// TwinCAT 3 PLC project IntelligenteWZM_PLCProject
// ProgramVersion: 3.1.4022.4
// libraries:
//   Tc2_Standard, * (Beckhoff Automation GmbH)
//   Tc2_System, * (Beckhoff Automation GmbH)
//   Tc2_Utilities, * (Beckhoff Automation GmbH)
//   Tc3_CM, * (Beckhoff Automation GmbH)
//   Tc3_CM_Base, * (Beckhoff Automation GmbH)
//   Tc3_Module, * (Beckhoff Automation GmbH)
//   Tc3_MultiArray, * (Beckhoff Automation GmbH)
//   VisuDialogs, * (System)
//   VisuSymbols,3.5.10.0,System
// project tree:
//   DUTs/ AdasConfiguration.TcDUT, AdasData_In.TcDUT, AdasSetup_Out.TcDUT, AdasStreamData.TcDUT, AdasStreamSetup.TcDUT, bsp.TcDUT, DW_TO_REAL.TcDUT, DW_TO_REAL_1.TcDUT, eAdasKom_State.TcDUT, eAdasKonfig_State.TcDUT, E_AnalysisIDs.TcDUT, sCCDataStreamHeader.TcDUT, sCCDataStreamSetup.TcDUT, Signalbezeichnungen.TcDUT, uCCDatagram.TcDUT
//   DUTs/Error Monitoring/ ST_HRErrHist.TcDUT
//   DUTs/Function Generator/ E_FunctionType.TcDUT
//   / GlobalTextList.TcGTLO, PlcTask.TcTTO, Visualization Manager.TcVMO (not stored)
//   GVLs/ GVarL.TcGVL, GVL.TcGVL
//   POUs/ ADAS_Kom.TcPOU, ANALOG_INPUT_EL3104.TcPOU (not stored), ANALOG_OUTPUT_EL4134.TcPOU, DATAMODULE.TcPOU, DATA_PREPARATION.TcPOU, DEFLECTION_CONTROL_FEED.TcPOU (not stored), DEFLECTION_CONTROL_POSITION.TcPOU, DP_CONFIG_IN_EL6731.TcPOU, DP_CONFIG_OUT_EL6731.TcPOU (not stored), ELLIP_FILTER.TcPOU, FORCE_SIGNALS.TcPOU, MAGNITUDESPECTRUM.TcPOU, MAIN.TcPOU, MAIN_CM.TcPOU, MEAS_STIFFNESS_COLLISION.TcPOU, MEAS_STIFFNESS_PROCESS.TcPOU, Test.TcPOU, TOUCH_PROBE_LINE.TcPOU (not stored), VARIABLES.TcGVL, SENSOR_CONTROL_EL6751.TcPOU (not stored), SENSOR_SIGNALS_EL6751.TcPOU (not stored)
//   POUs/Error Monitoring/ FB_HRErrHist.TcPOU
//   POUs/Function Generator/ FB_FunctionGenerator.TcPOU
//   VISUs/ Datamodule.TcVIS, PICTURES.TcIPO (not stored), VISUALISATION_DEFLEC_CONTROL.TcVIS (not stored), VISUALISATION_EMO2017.TcVIS (not stored), VISUALISATION_SENSOR_CONTROL.TcVIS (not stored), VISUALISATION_STIFFNESS_COLLISION.TcVIS (not stored), VISUALISATION_STIFFNESS_PROCESS.TcVIS
// real-time tasks:
//   TASK PlcTask: cycle T#1ms, priority 20, ADS port 350
//   TASK Task 1: cycle T#10ms, priority 1, ADS port 301
//   TASK CM_Task: cycle T#5ms, priority 2, ADS port 351
// I/O:
//   DEVICE Device 2 (EtherCAT), AmsNetId 169.254.30.239.3.1
//     Term 1 (EK1100) [EK1100 EtherCAT Coupler (2A E-Bus)]
//       Term 2 (EL4134) [EL4134 4Ch. Ana. Output -10/+10V, 16bit]
//       Term 3 (EL3104) [EL3104 4Ch. Ana. Input +/-10V Diff.]
//       Term 4 (EL6731-0010) [EL6731-0010 PROFIBUS DP Slave]
//       Term 5 (EL6751) [EL6751 CANopen Master]
//       Term 6 (EL9512) [EL9512 Power supply terminal 12V]
//       Term 11 (EL9011) [EL9011 End Terminal]
//     Term 7 (EK1100) [EK1100 EtherCAT Coupler (2A E-Bus)]
//       Term 8 (EL3632) [EL3632 2Ch. IEPE Sensor]
//       Term 9 (EL3632) [EL3632 2Ch. IEPE Sensor]
//       Term 10 (EL3632) [EL3632 2Ch. IEPE Sensor]
//       Term 12 (EL9011) [EL9011 End Terminal]
//   DEVICE Device 1 (EL6731-0010), AmsNetId 169.254.30.239.2.1
//     PROFIBUS-Sinumerik (EL6731-0010) // Vendor: BECKHOFF Revision: Revision 2.00
//   DEVICE Device 3 (EL6751), AmsNetId 169.254.30.239.4.1
//     CAN-Sensors (CANopen Node)
// variable links:
//   IntelligenteWZM_PLCProject/IntelligenteWZM_PLCProject Instance <-> Device 1 (EL6731-0010)/PROFIBUS-Sinumerik (EL6731-0010)
//     PlcTask Inputs/ADAS_Kom.ADAS_IN <-> Module 10 (64 WORD Slave-In/Master-Out)/Inputs/64 WORD Slave-In/Master-Out_0_0
//     PlcTask Inputs/VARIABLES.DP_MOSI_WORD_{1..4} <-> Module {5..8} (1 WORD Slave-In/Master-Out)/Inputs/1 WORD Slave-In/Master-Out_0_0  (4 links)
//     PlcTask Outputs/ADAS_Kom.adasStreamSetup_OUT <-> Module 9 (8 BYTE Slave-Out/Master-In)/Outputs/8 BYTE Slave-Out/Master-In_1_0
//     PlcTask Outputs/VARIABLES.DP_MISO_WORD_{1..4} <-> Module {1..4} (1 WORD Slave-Out/Master-In)/Outputs/1 WORD Slave-Out/Master-In_1_0  (4 links)
//   IntelligenteWZM_PLCProject/IntelligenteWZM_PLCProject Instance <-> Device 2 (EtherCAT)/Term 7 (EK1100)/Term 10 (EL3632)
//     PlcTask Inputs/VARIABLES.A_OVERSAMPLING_INPUT_5[0] <-> Ch1 Sample 0/Ch1 Value
//     PlcTask Inputs/VARIABLES.A_OVERSAMPLING_INPUT_5[1] <-> Ch1 Sample 1/Ch1 Value
//     PlcTask Inputs/VARIABLES.A_OVERSAMPLING_INPUT_5[2] <-> Ch1 Sample 2/Ch1 Value
//     PlcTask Inputs/VARIABLES.A_OVERSAMPLING_INPUT_5[3] <-> Ch1 Sample 3/Ch1 Value
//     PlcTask Inputs/VARIABLES.A_OVERSAMPLING_INPUT_5[4] <-> Ch1 Sample 4/Ch1 Value
//     PlcTask Inputs/VARIABLES.A_OVERSAMPLING_INPUT_5[5] <-> Ch1 Sample 5/Ch1 Value
//     PlcTask Inputs/VARIABLES.A_OVERSAMPLING_INPUT_5[6] <-> Ch1 Sample 6/Ch1 Value
//     PlcTask Inputs/VARIABLES.A_OVERSAMPLING_INPUT_5[7] <-> Ch1 Sample 7/Ch1 Value
//     PlcTask Inputs/VARIABLES.A_OVERSAMPLING_INPUT_5[8] <-> Ch1 Sample 8/Ch1 Value
//     PlcTask Inputs/VARIABLES.A_OVERSAMPLING_INPUT_5[9] <-> Ch1 Sample 9/Ch1 Value
//     PlcTask Inputs/VARIABLES.A_OVERSAMPLING_INPUT_6[0] <-> Ch2 Sample 0/Ch2 Value
//     PlcTask Inputs/VARIABLES.A_OVERSAMPLING_INPUT_6[1] <-> Ch2 Sample 1/Ch2 Value
//     PlcTask Inputs/VARIABLES.A_OVERSAMPLING_INPUT_6[2] <-> Ch2 Sample 2/Ch2 Value
//     PlcTask Inputs/VARIABLES.A_OVERSAMPLING_INPUT_6[3] <-> Ch2 Sample 3/Ch2 Value
//     PlcTask Inputs/VARIABLES.A_OVERSAMPLING_INPUT_6[4] <-> Ch2 Sample 4/Ch2 Value
//     PlcTask Inputs/VARIABLES.A_OVERSAMPLING_INPUT_6[5] <-> Ch2 Sample 5/Ch2 Value
//     PlcTask Inputs/VARIABLES.A_OVERSAMPLING_INPUT_6[6] <-> Ch2 Sample 6/Ch2 Value
//     PlcTask Inputs/VARIABLES.A_OVERSAMPLING_INPUT_6[7] <-> Ch2 Sample 7/Ch2 Value
//     PlcTask Inputs/VARIABLES.A_OVERSAMPLING_INPUT_6[8] <-> Ch2 Sample 8/Ch2 Value
//     PlcTask Inputs/VARIABLES.A_OVERSAMPLING_INPUT_6[9] <-> Ch2 Sample 9/Ch2 Value
//   IntelligenteWZM_PLCProject/IntelligenteWZM_PLCProject Instance <-> Device 2 (EtherCAT)/Term 7 (EK1100)/Term 8 (EL3632)
//     PlcTask Inputs/VARIABLES.A_OVERSAMPLING_INPUT_1[0] <-> Ch1 Sample 0/Ch1 Value
//     PlcTask Inputs/VARIABLES.A_OVERSAMPLING_INPUT_1[1] <-> Ch1 Sample 1/Ch1 Value
//     PlcTask Inputs/VARIABLES.A_OVERSAMPLING_INPUT_1[2] <-> Ch1 Sample 2/Ch1 Value
//     PlcTask Inputs/VARIABLES.A_OVERSAMPLING_INPUT_1[3] <-> Ch1 Sample 3/Ch1 Value
//     PlcTask Inputs/VARIABLES.A_OVERSAMPLING_INPUT_1[4] <-> Ch1 Sample 4/Ch1 Value
//     PlcTask Inputs/VARIABLES.A_OVERSAMPLING_INPUT_1[5] <-> Ch1 Sample 5/Ch1 Value
//     PlcTask Inputs/VARIABLES.A_OVERSAMPLING_INPUT_1[6] <-> Ch1 Sample 6/Ch1 Value
//     PlcTask Inputs/VARIABLES.A_OVERSAMPLING_INPUT_1[7] <-> Ch1 Sample 7/Ch1 Value
//     PlcTask Inputs/VARIABLES.A_OVERSAMPLING_INPUT_1[8] <-> Ch1 Sample 8/Ch1 Value
//     PlcTask Inputs/VARIABLES.A_OVERSAMPLING_INPUT_1[9] <-> Ch1 Sample 9/Ch1 Value
//     PlcTask Inputs/VARIABLES.A_OVERSAMPLING_INPUT_2[0] <-> Ch2 Sample 0/Ch2 Value
//     PlcTask Inputs/VARIABLES.A_OVERSAMPLING_INPUT_2[1] <-> Ch2 Sample 1/Ch2 Value
//     PlcTask Inputs/VARIABLES.A_OVERSAMPLING_INPUT_2[2] <-> Ch2 Sample 2/Ch2 Value
//     PlcTask Inputs/VARIABLES.A_OVERSAMPLING_INPUT_2[3] <-> Ch2 Sample 3/Ch2 Value
//     PlcTask Inputs/VARIABLES.A_OVERSAMPLING_INPUT_2[4] <-> Ch2 Sample 4/Ch2 Value
//     PlcTask Inputs/VARIABLES.A_OVERSAMPLING_INPUT_2[5] <-> Ch2 Sample 5/Ch2 Value
//     PlcTask Inputs/VARIABLES.A_OVERSAMPLING_INPUT_2[6] <-> Ch2 Sample 6/Ch2 Value
//     PlcTask Inputs/VARIABLES.A_OVERSAMPLING_INPUT_2[7] <-> Ch2 Sample 7/Ch2 Value
//     PlcTask Inputs/VARIABLES.A_OVERSAMPLING_INPUT_2[8] <-> Ch2 Sample 8/Ch2 Value
//     PlcTask Inputs/VARIABLES.A_OVERSAMPLING_INPUT_2[9] <-> Ch2 Sample 9/Ch2 Value
//   IntelligenteWZM_PLCProject/IntelligenteWZM_PLCProject Instance <-> Device 2 (EtherCAT)/Term 7 (EK1100)/Term 9 (EL3632)
//     PlcTask Inputs/VARIABLES.A_OVERSAMPLING_INPUT_3[0] <-> Ch1 Sample 0/Ch1 Value
//     PlcTask Inputs/VARIABLES.A_OVERSAMPLING_INPUT_3[1] <-> Ch1 Sample 1/Ch1 Value
//     PlcTask Inputs/VARIABLES.A_OVERSAMPLING_INPUT_3[2] <-> Ch1 Sample 2/Ch1 Value
//     PlcTask Inputs/VARIABLES.A_OVERSAMPLING_INPUT_3[3] <-> Ch1 Sample 3/Ch1 Value
//     PlcTask Inputs/VARIABLES.A_OVERSAMPLING_INPUT_3[4] <-> Ch1 Sample 4/Ch1 Value
//     PlcTask Inputs/VARIABLES.A_OVERSAMPLING_INPUT_3[5] <-> Ch1 Sample 5/Ch1 Value
//     PlcTask Inputs/VARIABLES.A_OVERSAMPLING_INPUT_3[6] <-> Ch1 Sample 6/Ch1 Value
//     PlcTask Inputs/VARIABLES.A_OVERSAMPLING_INPUT_3[7] <-> Ch1 Sample 7/Ch1 Value
//     PlcTask Inputs/VARIABLES.A_OVERSAMPLING_INPUT_3[8] <-> Ch1 Sample 8/Ch1 Value
//     PlcTask Inputs/VARIABLES.A_OVERSAMPLING_INPUT_3[9] <-> Ch1 Sample 9/Ch1 Value
//     PlcTask Inputs/VARIABLES.A_OVERSAMPLING_INPUT_4[0] <-> Ch2 Sample 0/Ch2 Value
//     PlcTask Inputs/VARIABLES.A_OVERSAMPLING_INPUT_4[1] <-> Ch2 Sample 1/Ch2 Value
//     PlcTask Inputs/VARIABLES.A_OVERSAMPLING_INPUT_4[2] <-> Ch2 Sample 2/Ch2 Value
//     PlcTask Inputs/VARIABLES.A_OVERSAMPLING_INPUT_4[3] <-> Ch2 Sample 3/Ch2 Value
//     PlcTask Inputs/VARIABLES.A_OVERSAMPLING_INPUT_4[4] <-> Ch2 Sample 4/Ch2 Value
//     PlcTask Inputs/VARIABLES.A_OVERSAMPLING_INPUT_4[5] <-> Ch2 Sample 5/Ch2 Value
//     PlcTask Inputs/VARIABLES.A_OVERSAMPLING_INPUT_4[6] <-> Ch2 Sample 6/Ch2 Value
//     PlcTask Inputs/VARIABLES.A_OVERSAMPLING_INPUT_4[7] <-> Ch2 Sample 7/Ch2 Value
//     PlcTask Inputs/VARIABLES.A_OVERSAMPLING_INPUT_4[8] <-> Ch2 Sample 8/Ch2 Value
//     PlcTask Inputs/VARIABLES.A_OVERSAMPLING_INPUT_4[9] <-> Ch2 Sample 9/Ch2 Value
//   IntelligenteWZM_PLCProject/IntelligenteWZM_PLCProject Instance <-> Device 3 (EL6751)/CAN-Sensors (CANopen Node)
//     PlcTask Inputs/VARIABLES.CAN_SENSOR_{1..10} <-> Sensor ID {1..10}/Inputs/CAN_IN_MESSAGE_D{1..10}  (10 links)
//     PlcTask Outputs/VARIABLES.CAN_HUB <-> HUB Control ID 0/Outputs/CAN_OUT_MESSAGE_CONTROL

CONFIGURATION IntelligenteWZM_PLCProject
    RESOURCE PLC ON TwinCAT3
        TASK PlcTask(INTERVAL := T#1ms, PRIORITY := 20);
        PROGRAM MAIN WITH PlcTask : MAIN;
        PROGRAM ADAS_Kom WITH PlcTask : ADAS_Kom;
    END_RESOURCE
END_CONFIGURATION

// ---- DUTs/AdasConfiguration.TcDUT
TYPE AdasConfiguration :
STRUCT
	track: ARRAY[0..(gVarL.gVar_NumberOfAdasTracks - 1)] OF BYTE;
	signal: ARRAY[0..(gVarL.gVar_NumberOfAdasTracks - 1)] OF BYTE;
	axis: ARRAY[0..(gVarL.gVar_NumberOfAdasTracks - 1)] OF BYTE;
END_STRUCT
END_TYPE

// ---- DUTs/AdasData_In.TcDUT
TYPE AdasData_In :

UNION
	asBin: ARRAY[0..(((gVarL.gVar_NumberOfAdasTracks * 2) + 4) - 1)] OF WORD;
	asData: AdasStreamData;
END_UNION

END_TYPE

// ---- DUTs/AdasSetup_Out.TcDUT
TYPE AdasSetup_Out :

UNION
	asSetup: AdasStreamSetup;
	asBin: ARRAY[0..7] OF BYTE;
END_UNION

END_TYPE

// ---- DUTs/AdasStreamData.TcDUT
TYPE AdasStreamData :
STRUCT
	/// type of the data block sent ( always 0xF )
	blockType: USINT;
	/// length of the whole data block sent ( in bytes )
	blockLength: USINT;
	/// number of the data tracks sent
	numActTracks: USINT;
	/// receipt flag of new selection
	acceptFlag: SINT;
	/// actual communication cycle in micro seconds
	comCycle: UINT;
	/// always 0
	fillByte1: BYTE;
	/// always 0
	fillByte2: BYTE;
	Data: ARRAY[0..(gVarL.gVar_NumberOfAdasTracks - 1)] OF DINT;
END_STRUCT
END_TYPE

// ---- DUTs/AdasStreamSetup.TcDUT
TYPE AdasStreamSetup :
STRUCT
	blockType: USINT := 15;
	blockLength: USINT := 8;
	fillByte1: USINT;
	fillByte2: USINT;
	selectTrack: USINT;
	selectAxis: USINT;
	selectSignal: USINT;
	selectFlag: SINT;
END_STRUCT
END_TYPE

// ---- DUTs/bsp.TcDUT
TYPE bsp :

UNION
	a: ARRAY[0..3] OF BYTE;
	b: DINT;
END_UNION

END_TYPE

// ---- DUTs/DW_TO_REAL.TcDUT
TYPE DW_TO_REAL :

UNION
	IntAsWord: ARRAY[0..1] OF WORD;
	IntAsReal: REAL;
END_UNION

END_TYPE

// ---- DUTs/DW_TO_REAL_1.TcDUT
TYPE DW_TO_REAL_1 :
UNION
	IntAsWord : ARRAY[0..1] OF WORD;
	IntAsReal: REAL;
END_UNION
END_TYPE

// ---- DUTs/eAdasKom_State.TcDUT
{attribute 'qualified_only' := ''}
{attribute 'strict' := ''}
TYPE eAdasKom_State :
(
	WaitForNC,
	SetDefaultkonfig,
	Running,
	Error
);
END_TYPE

// ---- DUTs/eAdasKonfig_State.TcDUT
{attribute 'qualified_only' := ''}
{attribute 'strict' := ''}
TYPE eAdasKonfig_State :
(
	Init,
	SendTrackConfig,
	WaitForSelectFlag,
	ConfigCurrent
);
END_TYPE

// ---- DUTs/Error Monitoring/ST_HRErrHist.TcDUT
TYPE ST_HRErrHist :
STRUCT
{attribute 'displaymode':='hex'}
	hrErrCode	: HRESULT;
	sErrSource	: STRING(63);
	nErrCount	: UDINT;
END_STRUCT
END_TYPE

// ---- DUTs/E_AnalysisIDs.TcDUT
TYPE E_AnalysisIDs :
(
	(* analysis chain *)
	eID_Source := 1,
	eID_MagSpec,
	eID_PowSpec,
	eID_SinkMag,
	eID_SinkPow
	//eID_Spectrum,
	//eID_Sink
	
) UDINT;
END_TYPE

// ---- DUTs/Function Generator/E_FunctionType.TcDUT
{attribute 'qualified_only'}
TYPE E_FunctionType :
(
	Sine,		// typical for vibrations originating from rotating machine
	Square,		// mixed sine signals good for analyzing spectrum
	Pulse,		// mixed sine signals good for analyzing spectrum
	Triangular,	// mixed sine signals good for analyzing spectrum
	Sawtooth,	// ramp-type vibrations, continuously increasing
	AM			// amplitude modulation: typical for vibrations originating from gear-tooth failure or bearing faults
);
END_TYPE

// ---- DUTs/sCCDataStreamHeader.TcDUT
TYPE sCCDataStreamHeader :
STRUCT
	byBlockType: BYTE;
	byBlockLength: BYTE;
	byNumActTracks: BYTE;
	byAcceptFlag: BYTE;
	uiComCycle: UINT;
	byFillByte1: BYTE;
	uiFillByte2: BYTE;
	aValue: ARRAY[0..29] OF DINT;
END_STRUCT
END_TYPE

// ---- DUTs/sCCDataStreamSetup.TcDUT
TYPE sCCDataStreamSetup :
STRUCT
	byBlockType: BYTE;
	byBlockLength: BYTE;
	byFillByte1: BYTE;
	byFillByte2: BYTE;
	bySelectTrack: BYTE;
	bySelectAxis: BYTE;
	bySelectSignal: BYTE;
	bySelectFlag: BYTE;
END_STRUCT
END_TYPE

// ---- DUTs/Signalbezeichnungen.TcDUT
TYPE Signalbezeichnungen :
STRUCT
	Name: STRING;
END_STRUCT
END_TYPE

// ---- DUTs/uCCDatagram.TcDUT
TYPE uCCDatagram :

UNION
	CCDataStreamHeader: sCCDataStreamHeader;
	CCData: ARRAY[0..63] OF WORD;
END_UNION

END_TYPE

// ---- GVLs/GVarL.TcGVL
VAR_GLOBAL
	///ADAS 
	iSignalID: ARRAY[0..20] OF BYTE;
	iAchseID: ARRAY[0..20] OF BYTE;
	iComCylce: BYTE := 20;
	iMode: INT := 10;
	iTracks: UINT;
	///Position x
	X_Machine_CS AT %Q*: LREAL;
	///Position y
	Y_Machine_CS AT %Q*: LREAL;
	///Position z
	Z_Machine_CS AT %Q*: LREAL;
	///Position c
	C_Machine_CS AT %Q*: LREAL;
	///Position b
	B_Machine_CS AT %Q*: LREAL;
	///Soll-Position x
	X_Machine_CS_soll AT %Q*: LREAL;
	///Geschwindigkeit x
	X_V_Machine_CS AT %Q*: LREAL;
	///Geschwindigkeit y
	Y_V_Machine_CS AT %Q*: LREAL;
	///Geschwindigkeit z
	Z_V_Machine_CS AT %Q*: LREAL;
	///Geschwindigkeit c
	C_V_Machine_CS AT %Q*: LREAL;
	///Geschwindigkeit b
	B_V_Machine_CS AT %Q*: LREAL;
	///Drehzahl n
	n_Spindle AT %Q*: LREAL;
	///Beschleunigung x
	X_a_Machine_CS AT %Q*: LREAL;
	///Beschleunigung y
	Y_a_Machine_CS AT %Q*: LREAL;
	///Beschleunigung z
	Z_a_Machine_CS AT %Q*: LREAL;
	///Beschleunigung c
	C_a_Machine_CS AT %Q*: LREAL;
	///Beschleunigung b
	B_a_Machine_CS AT %Q*: LREAL;
	///Strom x
	X_I AT %Q*: LREAL;
	///Strom y
	Y_I AT %Q*: LREAL;
	///Strom z
	Z_I AT %Q*: LREAL;
	///Strom c
	C_I AT %Q*: LREAL;
	///Strom b
	B_I AT %Q*: LREAL;
	///Strom Spindel
	n_I AT %Q*: LREAL;
	Data: uCCDatagram;
	///CCDataStreamSetupOUT 	 		:sCCDataStreamSetup;
	CCDataStreamSetupOUT AT %Q*: sCCDataStreamSetup;
	bGO: BOOL;

END_VAR

VAR_GLOBAL CONSTANT
	///ADAS
	gVar_NumberOfAdasTracks: INT := 30;
END_VAR

// ---- GVLs/GVL.TcGVL
VAR_GLOBAL CONSTANT
		MAX_BUFFER_SIZE : UDINT := 300;
		// Global variable for the MagnitudeSpectrum 
		cOversamples 	: UDINT 	:= 10;		// number of oversamples
		//cMaxChannels	: UDINT		:= 6; 		// number of the channel of the oversampling sensors
		cWindowLength	: UDINT		:= 3200;	// internal buffer size with 50% overlapping
		cBufferLength	: UDINT		:= cWindowLength/2;;	// buffer size
		
		cFFTLength		: UDINT		:= 4096;	// length of FFT for mag. spectrum	
		cFFTResult 		: UDINT 	:= cFFTLength/2+1;	// result of mag. spectrum (cFFTLength/2+1)
		cSamplingRate 	: UDINT		:= 10000; // Samplingrate of input signale(Accelerationssignal)
		
	
			
//		cFFTLength		: UDINT		:= 2048;				  // length of FFT 
//		cWindowLength   : UDINT     := 1800;				  // window length
//		cBufferLength	: UDINT		:= cWindowLength/2;	      // buffer size
//		cFFTResult 		: UDINT 	:= cFFTLength/2+1;		  // result of mag. spectrum - cFFTLength/2+1

	// Scenario 1:  Scaling such that amplitde of spectrum at MAIN.fSetFrequency should be MAIN.fSetAmplitude.
	//              Due to scalloping losses this is not exactly the case. 
	//              E.g. MAIN.fSetFrequency = 200 Hz -> Magnitude Spectrum peak = 12,989... ; Power Spectrum peak is squared value 12,989^2
	//              E.g. set MAIN.fSetFrequency = 185 Hz -> Magnitude Spectrum peak = 12,918... ; Power Spectrum peak is squared value 12,989^2    										 

		cDecibelScale   : BOOL      := FALSE;
		cScaling        : E_CM_ScalingType := eCM_PeakAmplitude;

	// Scenario 2: both spectra (power- and magnitude spectrum) are identical, due to decibel scaling!

	// cDecibelScale   : BOOL      := TRUE;
	// cScaling        : E_CM_ScalingType := eCM_PeakAmplitude;	

	// Scenario 3: Scaling such that summation over frequency bins is related to RMS value, in sine case MAIN.fSetAmplitude/sqrt(2) = 9.1924
	//             see Scaling Options for equations and line 57ff of MAIN POU for details.  
	
	// cDecibelScale   : BOOL      := FALSE;
	// cScaling        : E_CM_ScalingType := eCM_RMS;
		
END_VAR

// ---- POUs/VARIABLES.TcGVL
//{attribute 'qualified_only'}
VAR_GLOBAL
	// Eingangssignale aus den Klemmen 
	// Oversampling-Klemmen EL3632
	A_OVERSAMPLING_INPUT_1 AT%I*: ARRAY[0..9] OF INT; // Sensor 1 X 
	A_OVERSAMPLING_INPUT_2 AT%I*: ARRAY[0..9] OF INT; // Sensor 1 Y
	A_OVERSAMPLING_INPUT_3 AT%I*: ARRAY[0..9] OF INT; // Sensor 1 Z
	A_OVERSAMPLING_INPUT_4 AT%I*: ARRAY[0..9] OF INT; // Sensor 2 X
	A_OVERSAMPLING_INPUT_5 AT%I*: ARRAY[0..9] OF INT; // Sensor 2 Y
	A_OVERSAMPLING_INPUT_6 AT%I*: ARRAY[0..9] OF INT; // Sensor 2 Z
	
	//  CAN-BUS I/O (EL6751)
	CAN_HUB AT %Q*: ARRAY [0..7] OF USINT := [0, 0, 0, 0, 0, 0, 0, 0];		// HUB OUT FRAME, EVENT TIME HAS TO BE SET TO 65000!!!!
	CAN_SENSOR_1 AT %I*: CANMESSAGE;										// IN FRAME OF SENSOR ID 1
	CAN_SENSOR_2 AT %I*: CANMESSAGE;										// IN FRAME OF SENSOR ID 2
	CAN_SENSOR_3 AT %I*: CANMESSAGE;										// IN FRAME OF SENSOR ID 3
	CAN_SENSOR_4 AT %I*: CANMESSAGE;										// IN FRAME OF SENSOR ID 4
	CAN_SENSOR_5 AT %I*: CANMESSAGE;										// IN FRAME OF SENSOR ID 5
	CAN_SENSOR_6 AT %I*: CANMESSAGE;										// IN FRAME OF SENSOR ID 6
	CAN_SENSOR_7 AT %I*: CANMESSAGE;										// IN FRAME OF SENSOR ID 7
	CAN_SENSOR_8 AT %I*: CANMESSAGE;										// IN FRAME OF SENSOR ID 8
	CAN_SENSOR_9 AT %I*: CANMESSAGE;										// IN FRAME OF SENSOR ID 9
	CAN_SENSOR_10 AT %I*: CANMESSAGE;										// IN FRAME OF SENSOR ID 10
	
//	VARIABLES FOR SENSOR CONTROL (CAN)
	HUB_STATE: BOOL:=FALSE;													// TRUE: HUB IS SENDING FRAMES, FALSE: HUS IS NOT SENDING FRAMES  
	CAN_CONTROL_STATE: BYTE := 0;											// SENSOR COMMANDs, 0: STOP SENSOR, 1: START SENSOR, 2: RESET SENSOR, 3: PARAMETRIZE SENSOR, 11: DEFAULT 
	CAN_TRIGGER_STATE: BYTE := 0;											// 1: SENSOR TRIGGER ON, 0: SENSOR TRIGGER OFF
	CAN_CONTROL_FRAME: ARRAY [0..7] OF USINT :=[0, 0, 0, 0, 0, 0, 0, 0];	// FRAME TO BE SENT BY THE HUB TO THE SENSORS
	CAN_PARAMETER_FRAME: ARRAY [0..7] OF USINT :=[0, 0, 0, 0, 0, 0, 0, 0];	// PARAMETER FRAME TO BE SENT BY THE HUB TO THE SENSORS
	K_TRIGGER: WORD:=1;														// SETTING FOR TRIGGER FREQUENCY, K_TRIGGER=T_Trigger/T_PLC
	M_PER_FRAME: USINT:=1;  												// NUMBER OF NEEDED MEASUREMENTS IN FRAME COMMING FROM SENSORS, M_PER_FRAME=1..4
	N_SAMPLES_PER_M: USINT:=1;												// NUMBER OF SAMPLES PER NEEDED MEASUREMENT
	SIGNAL_SYNCH: WORD;														// TRIGGER NUMBER FOR SIGNAL SYNCHRONISATION
	
//  VARIABLES FOR SENSOR SIGNALS	
	SIGNAL_SENSOR_1: ARRAY[1..5] OF WORD;									// SIGNALS FROM SENSOR ID 1, [1]..[4]: MEASUREMENT 1..4, [5]: COMBINED SIGNAL FROM MEASUREMENTS
	SIGNAL_SENSOR_2: ARRAY[1..5] OF WORD;									// SIGNALS FROM SENSOR ID 2, [1]..[4]: MEASUREMENT 1..4, [5]: COMBINED SIGNAL FROM MEASUREMENTS
	SIGNAL_SENSOR_3: ARRAY[1..5] OF WORD;									// SIGNALS FROM SENSOR ID 3, [1]..[4]: MEASUREMENT 1..4, [5]: COMBINED SIGNAL FROM MEASUREMENTS
	SIGNAL_SENSOR_4: ARRAY[1..5] OF WORD;									// SIGNALS FROM SENSOR ID 4, [1]..[4]: MEASUREMENT 1..4, [5]: COMBINED SIGNAL FROM MEASUREMENTS
	SIGNAL_SENSOR_5: ARRAY[1..5] OF WORD;									// SIGNALS FROM SENSOR ID 5, [1]..[4]: MEASUREMENT 1..4, [5]: COMBINED SIGNAL FROM MEASUREMENTS
	SIGNAL_SENSOR_6: ARRAY[1..5] OF WORD;									// SIGNALS FROM SENSOR ID 6, [1]..[4]: MEASUREMENT 1..4, [5]: COMBINED SIGNAL FROM MEASUREMENTS
	SIGNAL_SENSOR_7: ARRAY[1..5] OF WORD;									// SIGNALS FROM SENSOR ID 7, [1]..[4]: MEASUREMENT 1..4, [5]: COMBINED SIGNAL FROM MEASUREMENTS
	SIGNAL_SENSOR_8: ARRAY[1..5] OF WORD;									// SIGNALS FROM SENSOR ID 8, [1]..[4]: MEASUREMENT 1..4, [5]: COMBINED SIGNAL FROM MEASUREMENTS
	SIGNAL_SENSOR_9: ARRAY[1..5] OF WORD;									// SIGNALS FROM SENSOR ID 9, [1]..[4]: MEASUREMENT 1..4, [5]: COMBINED SIGNAL FROM MEASUREMENTS
	SIGNAL_SENSOR_10: ARRAY[1..5] OF WORD;									// SIGNALS FROM SENSOR ID 10, [1]..[4]: MEASUREMENT 1..4, [5]: COMBINED SIGNAL FROM MEASUREMENTS
	
	SIGNAL_SENSOR_1_FLT: REAL;												// FILTERED SIGNAL SIGNAL_SENSOR_1[5]
	SIGNAL_SENSOR_2_FLT: REAL;												// FILTERED SIGNAL SIGNAL_SENSOR_2[5]
	SIGNAL_SENSOR_3_FLT: REAL;												// FILTERED SIGNAL SIGNAL_SENSOR_3[5]
	SIGNAL_SENSOR_4_FLT: REAL;												// FILTERED SIGNAL SIGNAL_SENSOR_4[5]	
	SIGNAL_SENSOR_5_FLT: REAL;												// FILTERED SIGNAL SIGNAL_SENSOR_5[5]
	SIGNAL_SENSOR_6_FLT: REAL;												// FILTERED SIGNAL SIGNAL_SENSOR_6[5]
	SIGNAL_SENSOR_7_FLT: REAL;												// FILTERED SIGNAL SIGNAL_SENSOR_7[5]
	SIGNAL_SENSOR_8_FLT: REAL;												// FILTERED SIGNAL SIGNAL_SENSOR_8[5]
	SIGNAL_SENSOR_9_FLT: REAL;												// FILTERED SIGNAL SIGNAL_SENSOR_9[5]
	SIGNAL_SENSOR_10_FLT: REAL;												// FILTERED SIGNAL SIGNAL_SENSOR_10[5]
	
	
	// SETTINGS FOR LOW PASS FILTERS
	//Matlab: Fsamp=1000, Fg=10, Rp=0.5, Rs=20, Wp=Fg/Fsamp*2, [B_FILTER,A_FILTER] = ellip(3,Rp,Rs,Wp);
	//A=['[' num2str(A_FILTER(1)) ', ' num2str(A_FILTER(2)) ', ' num2str(A_FILTER(3)) ', ' num2str(A_FILTER(4)) ']']
	//B=['[' num2str(B_FILTER(1)) ', ' num2str(B_FILTER(2)) ', ' num2str(B_FILTER(3)) ', ' num2str(B_FILTER(4)) ']']
	A_FILTER: ARRAY [1..4] OF REAL:=[1, -2.8353, 2.6948, -0.85785];
	B_FILTER: ARRAY [1..4] OF REAL:=[0.021368, -0.020532, -0.020532, 0.021368];

	SENSOR_STATE: ARRAY[1..10] OF BOOL;										// TRUE: SENSOR IS SENSING FRAMES, FALSE: SENSOR IS NOT SENDING FRAMES
	SIGNAL_DEVIATION: ARRAY [1..10] OF WORD:=[0,0,0,0,0,0,0,0,0,0];			// NOISE DEVIATION OF SENSOR SIGNALS
	
	// 	PROFI-BUS I/O (EL6731)
	
	DP_MISO_WORD_1 AT %Q*: WORD;											// OUT FRAME 1 (BECKHOFF TO SINUMERIK)
	DP_MISO_WORD_2 AT %Q*: WORD;											// OUT FRAME 2 (BECKHOFF TO SINUMERIK)
	DP_MISO_WORD_3 AT %Q*: WORD;											// OUT FRAME 3 (BECKHOFF TO SINUMERIK)
	DP_MISO_WORD_4 AT %Q*: WORD;											// OUT FRAME 4 (BECKHOFF TO SINUMERIK)
	DP_MOSI_WORD_1 AT %I*: WORD;											// IN FRAME 1 (SINUMERIK TO BECKHOFF)
	DP_MOSI_WORD_2 AT %I*: WORD;											// IN FRAME 2 (SINUMERIK TO BECKHOFF)
	DP_MOSI_WORD_3 AT %I*: WORD;											// IN FRAME 3 (SINUMERIK TO BECKHOFF)
	DP_MOSI_WORD_4 AT %I*: WORD;											// IN FRAME 4 (SINUMERIK TO BECKHOFF)
	
//	ANALOG I (EL3104)
	A_INPUT_1 AT %I*: INT;													// ANALOG INPUT 1
	A_INPUT_2 AT %I*: INT;													// ANALOG INPUT 2
	A_INPUT_3 AT %I*: INT;													// ANALOG INPUT 3
	A_INPUT_4 AT %I*: INT;													// ANALOG INPUT 4

// Input fuer Beschleunigungssensoren	
	A_INPUT_5 	AT %I*: INT;													// ANALOG INPUT 5
	A_INPUT_6 	AT %I*: INT;													// ANALOG INPUT 6
	A_INPUT_7 	AT %I*: INT;													// ANALOG INPUT 6
	A_INPUT_8 	AT %I*: INT;													// ANALOG INPUT 6
	A_INPUT_9 	AT %I*: INT;													// ANALOG INPUT 6
	A_INPUT_10 	AT %I*: INT;													// ANALOG INPUT 6
	
//SETTINGS FOR GAINS
	A_GAIN_1: REAL:=-100;
	A_GAIN_2: REAL:=-100;
	A_GAIN_3: REAL:=-100;
	A_GAIN_4: REAL:=1;
	
//  ANALOG I SIGNALS
	A_SIGNAL_1 : REAL:=0;													// ANALOG INPUT SIGNAL 1 
	A_SIGNAL_2 : REAL:=0;													// ANALOG INPUT SIGNAL 2
	A_SIGNAL_3 : REAL:=0;													// ANALOG INPUT SIGNAL 3
	A_SIGNAL_4 : REAL:=0;													// ANALOG INPUT SIGNAL 4
	A_SIGNAL_5 : REAL:=0;
	A_SIGNAL_6 : REAL:=0;
	A_SIGNAL_7 : REAL:=0;
	
//  VARIABLES FOR FORCE SIGNALS
	SIGNAL_FORCE: ARRAY[1..3] OF REAL;										// FORCE SIGNALS, 1: X-FORCE, 2: Y-FORCE, 3: Z-FORCE in MCS
	SIGNAL_FORCE_FLT: ARRAY[1..3] OF REAL;									// FILTERED FORCE SIGNALS, 1: X-FORCE, 2: Y-FORCE, 3: Z-FORCE in MCS
	FORCE_RESET: WORD :=0;													// CONTROL VARIABLE FOR FORCE RESET
	FORCE_ACT: REAL;														// ACTUAL USED FORCE SIGNAL 

//	VARIABLES FOR POSITION SIGNALS
	Y_POSITION_ACT: REAL;
	X_POSITION_ACT: REAL;
	Z_POSITION_ACT: REAL; 

	
// FORCE CALIBARTION MATRIXES
FC_MATRIX_X: ARRAY [1..10] OF REAL:=[-0.76798,0.10123,1.0077,-0.3399,0.8848,-1.162,0,1.0382];
FC_MATRIX_Y: ARRAY [1..10] OF REAL:=[-0.92845,0.11284,1.2124,-0.39371,0.99951,-1.3615,0,1.1904]; 
FC_MATRIX_Z: ARRAY [1..10] OF REAL:=[-0.30943,0.061409,0.43615,-0.13896,0.34508,-0.49067,0,0.43918];	
	
	//FC_MATRIX_X: ARRAY [1..10] OF REAL:=[0,0,0,0,0,1,0,0,0,-1];
	//FC_MATRIX_Y: ARRAY [1..10] OF REAL:=[0,0,0,0,0,1,0,0,0,-1]; 
	//FC_MATRIX_Z: ARRAY [1..10] OF REAL:=[0,0,0,0,0,0,0,0,0,0];
	
	

	
//  VARIABLES FROM NC PROGRAM 	
	ACT_NC_PROGRAM: WORD:=0;												
	ACT_NC_PROGRAM_STEP: WORD:=0;												
	ACT_NC_PARAM_3: WORD:=0;
	ACT_NC_PARAM_4: WORD:=0;
	ACT_NC_PARAM_5: REAL:=0;
	ACT_NC_PARAM_6: REAL:=0;
	
//	VARIABLES TO NC PROGRAM
	SET_NC_PARAM_1: WORD:=0;
	SET_NC_PARAM_2: WORD:=0;
	SET_NC_PARAM_3: WORD:=0;
	SET_NC_PARAM_4: WORD:=0;
	
	
//  VARIABLES FOR TOOL STIFFNESS MEASUREMENT	
	TOOL_STIFFNESS : ARRAY [1..2] OF REAL:=[0, 0];				// in N/µm FFOR CONTACT PTS
	COLLISION_DISTANCE : REAL:=0;			// in µm
	SHAPE_DEVIATION : REAL:=0;				// in µm
	FORCE_DEVIATION : ARRAY [1..2] OF REAL:=[0, 0];				// in N
	TOOL_BLENDING_STIFFNESS : ARRAY [1..2] OF REAL:=[0, 0];		// in N.mm²
	TOOL_LENGTH : REAL:=33; 				// in mm
	Z_POS_STIFF_MEAS : ARRAY [1..2] OF REAL:=[0, 0]; 			// in mm
	a_POS : ARRAY [1..2] OF REAL:=[0, 0];						// in mm

	TOOL_STIFFNESS_SELC_PTS: ARRAY [1..2, 1..5] OF REAL:=[0, 0, 8, 0, 0, 0, 0, 8, 0, 0];
	Z_POS_SELC_PTS: ARRAY [1..5] OF REAL:=[0, -2.5, -8.5, -12, -17];
	a_REF: REAL:=0;
	AX_SELC_PTS: ARRAY [1..5] OF REAL:=[0, 0, 0, 0, 0];
	Z_POS_REF: REAL:=-17;
	
	TOOL_STIFFNESS_ACT: REAL:=0;
	TOOL_BLENDING_STIFFNESS_ACT: REAL:=0;
	a_ACT: REAL:=0;
	AX_ACT: REAL:=0;
	Z_POS_ACT: REAL:=0;
	
	
	
	
//  VARIABLES FOR TOOL DEFLECTION CONTROL 
	DEFLECTION_ACT: REAL;
	DEFLECTION_REF: REAL:=25;
	DEFLECTION_DIF: REAL:=0;
	DEFLECTION_DIF_SUM: REAL:=0;
	DEFLECTION_CONTROL_ON: INT:=0;	
	CONTROL_RESET: INT:=0;	
	CONTROLLER_TYPE: INT:=0;
	CONTROL_START_CONDITION: BOOL:=FALSE;
	CONTROL_START: INT:=0;
	CUTTING_ON: INT:=0;	
	CUTTING_FORCE_MIN: REAL:=50;
	REF_REACHED: INT:=0;
	
	SATURATION_OVRD_MAX: REAL:=120;
	SATURATION_OVRD_MIN: REAL:=20;
	OVRD_MID: REAL:=70;	
	OVRD_MACHINE: REAL:=100;
	OVRD_REG: REAL:=0;
	OVRD_REG_P: REAL:=0;
	OVRD_REG_I: REAL:=0;
	WINDUP: REAL:=0;
	OVRD_DIF: REAL;
	K_P: REAL:=0.75;								// PROPORTIONAL REGULATOR FACTOR
	K_I: REAL:=60;						// INT. REGULATOR FACTOR
	T_S: REAL:=0.004;							// SAMPLE TIME
	K_WINDUP: REAL:=0.05;						// WINDUP FACTOR
	
	
	SATURATION_POS_MAX: REAL:=200;
	SATURATION_POS_MIN: REAL:=-200;
	POS_MID: REAL:=0;	
	POS_MACHINE: REAL:=0;
	POS_REG: REAL:=0;
	POS_REG_P: REAL:=0;
	POS_REG_I: REAL:=0;
	POS_WINDUP: REAL:=0;
	POS_DIF: REAL;
	POS_K_P: REAL:=1;//0.5625;								// PROPORTIONAL REGULATOR FACTOR
	POS_K_I: REAL:=0;//10;//4.563;							// INT. REGULATOR FACTOR
	POS_T_S: REAL:=0.004;							// SAMPLE TIME
	POS_K_WINDUP: REAL:=0;						// WINDUP FACTOR
	

//  VARIABLES FOR TOUCH PROBE LINE
	PTS_POSITION: 		ARRAY[1..50] OF REAL;
	PTS_MEASUREMENT: 		ARRAY[1..50] OF REAL;	
	PTS_SELCT_HISTOGRAM: ARRAY [1..10] OF WORD := [1, 2, 3, 4, 5, 6, 7, 8, 9, 10];
	PTS_MEASUREMENT_HISTOGRAM_1:  ARRAY [1..10] OF REAL;
	PTS_MEASUREMENT_HISTOGRAM_2:  ARRAY [1..10] OF REAL;
	RESULT: ARRAY [0..1] OF REAL:=[0,0];
	VarTest: BOOL := TRUE;
	
	Test_Var: WORD:=0;
	
	
	
	
END_VAR

// ---- POUs/MAIN.TcPOU
PROGRAM MAIN
VAR_INPUT
//ADAS
	ADAS_in		AT %I* 	: ARRAY[0..63] OF WORD; //ADAS_Rohdaten
END_VAR


IF FORCE_RESET=1 THEN
	RESULT[0]:=0;
	PTS_MEASUREMENT_HISTOGRAM_2[2]:=0;
	RESULT[1]:=0;
END_IF

IF VarTest = TRUE THEN
	VarTest := FALSE;
END_IF

IF VarTest = FALSE THEN
	VarTest := TRUE;
END_IF

ANALOG_INPUT_EL3104();
//ANALOG_OUTPUT_EL4134();
DP_CONFIG_IN_EL6731();
SENSOR_CONTROL_EL6751();
SENSOR_SIGNALS_EL6751();
FORCE_SIGNALS();
//Test();
DATAMODULE();

MEAS_STIFFNESS_COLLISION();
MEAS_STIFFNESS_PROCESS();
DEFLECTION_CONTROL_FEED();
DEFLECTION_CONTROL_POSITION();
TOUCH_PROBE_LINE();
DP_CONFIG_OUT_EL6731();


//ADAS Daten
	//x-Achse (soll alles stimmen)
X_Machine_CS 		:= DINT_TO_LREAL(ADAS_Kom.adasData[1])	/ 10000; //Umrechnung in: mm -> /10000 (10000 inkremente sind 1mm)
X_Machine_CS_soll 	:= DINT_TO_LREAL(ADAS_Kom.adasData[27])	/ 10000; //Umrechnung in: mm -> /10000 (10000 inkremente sind 1mm)
X_V_Machine_CS 		:= DINT_TO_LREAL(ADAS_Kom.adasData[6])	/ 10000; //Umrechnung in: mm/s-> /10000
X_a_Machine_CS 		:= DINT_TO_LREAL(ADAS_Kom.adasData[12])	/ 10000; //Umrechnung in: mm/s²-> /10000
X_I					:= DINT_TO_LREAL(ADAS_Kom.adasData[18])	/ 1000;  //Umrechnung in: A -> /1000

	//y-Achse  (soll alles stimmen)
Y_Machine_CS 		:= DINT_TO_LREAL(ADAS_Kom.adasData[2]) 	/ 10000; //Umrechnung in: mm -> /10000
Y_V_Machine_CS 		:= DINT_TO_LREAL(ADAS_Kom.adasData[7]) 	/ 10000; //Umrechnung in: mm/s-> /10000
Y_a_Machine_CS 		:= DINT_TO_LREAL(ADAS_Kom.adasData[13])	/ 10000; //Umrechnung in: mm/s²-> /10000
Y_I					:= DINT_TO_LREAL(ADAS_Kom.adasData[19])	/ 1000;  //Umrechnung in: A -> /1000
	//z-Achse (soll alles stimmen)
Z_Machine_CS 		:= DINT_TO_LREAL(ADAS_Kom.adasData[3]) 	/ 10000; //Umrechnung in: mm -> /10000
Z_V_Machine_CS 		:= DINT_TO_LREAL(ADAS_Kom.adasData[8]) 	/ 10000; //Umrechnung in: mm/s-> /10000
Z_a_Machine_CS 		:= DINT_TO_LREAL(ADAS_Kom.adasData[14])	/ 10000; //Umrechnung in: mm/s²-> /10000
Z_I					:= DINT_TO_LREAL(ADAS_Kom.adasData[20])	/ 1000;  //Umrechnung in: A -> /1000
	//C-Achse (soll alles stimmen)
C_Machine_CS 		:= DINT_TO_LREAL(ADAS_Kom.adasData[4] 	MOD 3600000)/ 10000 ; //Umrechnung in: mm -> /10000
C_V_Machine_CS 		:= DINT_TO_LREAL(ADAS_Kom.adasData[9]) 	/ 10000; //Umrechnung in: mm/s-> /10000
C_a_Machine_CS 		:= DINT_TO_LREAL(ADAS_Kom.adasData[15])	/ 10000; //Umrechnung in: mm/s²-> /10000
C_I 				:= DINT_TO_LREAL(ADAS_Kom.adasData[21])	/ 1000;  //Umrechnung in: A -> /1000
	//B-Achse (B_Machine_CS wid von Spinel beschrieben)
B_Machine_CS		:= DINT_TO_LREAL(ADAS_Kom.adasData[24]) / 10000; //Umrechnung in: mm -> /10000 //b
B_V_Machine_CS 		:= DINT_TO_LREAL(ADAS_Kom.adasData[10]) / 10000; //Umrechnung in: mm/s-> /10000
B_a_Machine_CS 		:= DINT_TO_LREAL(ADAS_Kom.adasData[16]) / 10000; //Umrechnung in: mm/s²-> /10000
B_I 				:= DINT_TO_LREAL(ADAS_Kom.adasData[22]) / 1000;  //Umrechnung in: A -> /1000
	//Spindel
n_Spindle 			:= (DINT_TO_LREAL(ADAS_Kom.adasData[5])/360)*60/10000 ; //kommt in milli°/s Umrechnung in: 1/min-> *0,166667
n_I 				:= DINT_TO_LREAL(ADAS_Kom.adasData[23])/1000; //Umrechnung in: A -> /1000

END_PROGRAM

// ---- POUs/DP_CONFIG_IN_EL6731.TcPOU
PROGRAM DP_CONFIG_IN_EL6731
VAR
	UNION_DW2REAL_1 : DW_TO_REAL;	
	UNION_DW2REAL_2: DW_TO_REAL;	
END_VAR

ACT_NC_PROGRAM:=DP_MOSI_WORD_1;													
ACT_NC_PROGRAM_STEP:=DP_MOSI_WORD_2;	
ACT_NC_PARAM_3:=DP_MOSI_WORD_3;	
ACT_NC_PARAM_4:=DP_MOSI_WORD_4;	
UNION_DW2REAL_1.IntAsWord[0] := DP_MOSI_WORD_3;	
UNION_DW2REAL_1.IntAsWord[1] := DP_MOSI_WORD_4;	
ACT_NC_PARAM_5:= UNION_DW2REAL_1.IntAsReal;

UNION_DW2REAL_2.IntAsWord[0] := DP_MOSI_WORD_1;	
UNION_DW2REAL_2.IntAsWord[1] := DP_MOSI_WORD_2;	
ACT_NC_PARAM_6:= UNION_DW2REAL_2.IntAsReal;

END_PROGRAM

// ---- POUs/FORCE_SIGNALS.TcPOU
PROGRAM FORCE_SIGNALS
VAR
	RESET_FORCE_VAL: ARRAY[1..3] OF REAL := [0,0,0];
	FORCE_ROW: ARRAY[1..3] OF REAL;
	FORCE_SUM: ARRAY[1..3] OF REAL:= [0,0,0];
	INK: INT:=0;
	
	FILTER_FX:ELLIP_FILTER;
	FILTER_FY:ELLIP_FILTER;
	FILTER_FZ:ELLIP_FILTER;
	
	
END_VAR

FORCE_ROW[1]:=(FC_MATRIX_X[1]*SIGNAL_SENSOR_1[1]+FC_MATRIX_X[2]*SIGNAL_SENSOR_2[1]+FC_MATRIX_X[3]*SIGNAL_SENSOR_3[1]+FC_MATRIX_X[4]*SIGNAL_SENSOR_4[1]+FC_MATRIX_X[5]*SIGNAL_SENSOR_5[1]+FC_MATRIX_X[6]*SIGNAL_SENSOR_6[1]+FC_MATRIX_X[7]*SIGNAL_SENSOR_7[1]+FC_MATRIX_X[8]*SIGNAL_SENSOR_8[1]+FC_MATRIX_X[9]*SIGNAL_SENSOR_9[1]+FC_MATRIX_X[10]*SIGNAL_SENSOR_10[1]);
FORCE_ROW[2]:=(FC_MATRIX_Y[1]*SIGNAL_SENSOR_1[1]+FC_MATRIX_Y[2]*SIGNAL_SENSOR_2[1]+FC_MATRIX_Y[3]*SIGNAL_SENSOR_3[1]+FC_MATRIX_Y[4]*SIGNAL_SENSOR_4[1]+FC_MATRIX_Y[5]*SIGNAL_SENSOR_5[1]+FC_MATRIX_Y[6]*SIGNAL_SENSOR_6[1]+FC_MATRIX_Y[7]*SIGNAL_SENSOR_7[1]+FC_MATRIX_Y[8]*SIGNAL_SENSOR_8[1]+FC_MATRIX_Y[9]*SIGNAL_SENSOR_9[1]+FC_MATRIX_Y[10]*SIGNAL_SENSOR_10[1]);
FORCE_ROW[3]:=(FC_MATRIX_Z[1]*SIGNAL_SENSOR_1[1]+FC_MATRIX_Z[2]*SIGNAL_SENSOR_2[1]+FC_MATRIX_Z[3]*SIGNAL_SENSOR_3[1]+FC_MATRIX_Z[4]*SIGNAL_SENSOR_4[1]+FC_MATRIX_Z[5]*SIGNAL_SENSOR_5[1]+FC_MATRIX_Z[6]*SIGNAL_SENSOR_6[1]+FC_MATRIX_Z[7]*SIGNAL_SENSOR_7[1]+FC_MATRIX_Z[8]*SIGNAL_SENSOR_8[1]+FC_MATRIX_Z[9]*SIGNAL_SENSOR_9[1]+FC_MATRIX_Z[10]*SIGNAL_SENSOR_10[1]);

IF FORCE_RESET>0 THEN
	FORCE_SUM[1]:=FORCE_ROW[1]+FORCE_SUM[1];
	FORCE_SUM[2]:=FORCE_ROW[2]+FORCE_SUM[2];
	FORCE_SUM[3]:=FORCE_ROW[3]+FORCE_SUM[3];
	INK:=INK+1;
	IF INK=1000 THEN
		RESET_FORCE_VAL[1]:=FORCE_SUM[1]/INK;
		RESET_FORCE_VAL[2]:=FORCE_SUM[2]/INK;
		RESET_FORCE_VAL[3]:=FORCE_SUM[3]/INK;
		INK:=0;
		FORCE_RESET:=0;
		FORCE_SUM[1]:=0;
		FORCE_SUM[2]:=0;
		FORCE_SUM[3]:=0;
	END_IF
END_IF


SIGNAL_FORCE[1]:=FORCE_ROW[1]-RESET_FORCE_VAL[1];
SIGNAL_FORCE[2]:=FORCE_ROW[2]-RESET_FORCE_VAL[2];
SIGNAL_FORCE[3]:=FORCE_ROW[3]-RESET_FORCE_VAL[3];

FILTER_FX(ssMethodType:=1 , IN:= SIGNAL_FORCE[1], OUT=> SIGNAL_FORCE_FLT[1]);
FILTER_FY(ssMethodType:=1 , IN:= SIGNAL_FORCE[2], OUT=> SIGNAL_FORCE_FLT[2]);
FILTER_FZ(ssMethodType:=1 , IN:= SIGNAL_FORCE[3], OUT=> SIGNAL_FORCE_FLT[3]);

END_PROGRAM

// ---- POUs/ELLIP_FILTER.TcPOU
FUNCTION_BLOCK ELLIP_FILTER
VAR_INPUT
	ssMethodType: SINT;
	IN: LREAL;
END_VAR
VAR_OUTPUT
	OUT: LREAL;
END_VAR
VAR
	DiscreteFilter_tmp: LREAL;
	DiscreteFilter_states: ARRAY[0..2] OF LREAL;
END_VAR



CASE ssMethodType OF
    0: 
        

        (* InitializeConditions for DiscreteFilter: '<S1>/Discrete Filter' *)
        DiscreteFilter_states[0] := 0.0;
        DiscreteFilter_states[1] := 0.0;
        DiscreteFilter_states[2] := 0.0;
		
    1: 
        

        (* DiscreteFilter: '<S1>/Discrete Filter' incorporates:
         *  Inport: '<Root>/IN' *)
        DiscreteFilter_tmp := (((IN - (A_FILTER[2] * DiscreteFilter_states[0])) - (A_FILTER[3] * DiscreteFilter_states[1])) - (A_FILTER[4] * DiscreteFilter_states[2])) / A_FILTER[1];
        

        (* Outport: '<Root>/OUT' incorporates:
         *  DiscreteFilter: '<S1>/Discrete Filter' *)
        OUT := (((B_FILTER[1] * DiscreteFilter_tmp) + (B_FILTER[2] * DiscreteFilter_states[0])) + (B_FILTER[3] * DiscreteFilter_states[1])) + (B_FILTER[4] * DiscreteFilter_states[2]);
        

        (* Update for DiscreteFilter: '<S1>/Discrete Filter' *)
        DiscreteFilter_states[2] := DiscreteFilter_states[1];
        DiscreteFilter_states[1] := DiscreteFilter_states[0];
        DiscreteFilter_states[0] := DiscreteFilter_tmp;
END_CASE;

END_FUNCTION_BLOCK

// ---- POUs/DATAMODULE.TcPOU
PROGRAM DATAMODULE
VAR
	//ADAS-Daten (Spindelstrom, Achspositionen und Drehzahl) aus GVL, dann kann es weg?
	X_Machine_CS 	: LREAL;
	Y_Machine_CS 	: LREAL;
	Z_Machine_CS 	: LREAL;
	C_Machine_CS 	: LREAL;
	B_Machine_CS 	: LREAL;

	X_V_Machine_CS 	: LREAL;
	Y_V_Machine_CS 	: LREAL;
	Z_V_Machine_CS 	: LREAL;
	C_V_Machine_CS 	: LREAL;
	B_V_Machine_CS 	: LREAL;
	n_Spindle 		: LREAL;
	
	X_a_Machine_CS 	: LREAL;
	Y_a_Machine_CS 	: LREAL;
	Z_a_Machine_CS 	: LREAL;
	C_a_Machine_CS 	: LREAL;
	B_a_Machine_CS 	: LREAL;
	n_a_Spindle 	: LREAL;
	
	X_I				: LREAL;
	Y_I				: LREAL;
	Z_I				: LREAL;
	C_I				: LREAL;
	B_I 			: LREAL;
	n_I 			: LREAL;
			
	
	//VARIABLEN FÜR SCHNITTSTELLEN:
	{attribute 'OPC.UA.DA' := '1'}
	Database :ARRAY[0..27]OF LREAL;

	
	//Für GUI
	yGraph1 : LREAL;
	yGraph2 : LREAL;
	yGraph3		: LREAL;
	Timer		: REAL := 0;
	//Parameter von GUI
	{attribute 'OPC.UA.DA' := '1'}
	Depth		: LREAL;
	{attribute 'OPC.UA.DA' := '1'}
	Width		: LREAL;
	Select_NN1	: BOOL;
	Select_NN2  : BOOL;
	Start  		: BOOL;
	Stop	  	: BOOL;
	Reset  		: BOOL;
	//für NN-Config-Info für die Vorverarbeitung
	{attribute 'OPC.UA.DA' := '1'}
	Config_NN1  : BOOL := FALSE;
	{attribute 'OPC.UA.DA' := '1'}
	Config_NN2  : BOOL := FALSE;
	{attribute 'OPC.UA.DA' := '1'}
	NewConfig	: BOOL := FALSE;
	//Configbestätigung von NN
	{attribute 'OPC.UA.DA' := '1'}
	{attribute 'OPC.UA.DA.Access' := '1'}
	AcceptConfig : BOOL;


	CycleTime		  : INT := 10; (*ms*)
	CommunicationState: INT; (*1=SendConfig, 2=WaitForConfig, 3=Start, 4=Stop, 5=Reset*)
	SetZeros : INT :=0;
	// Trigger Statusänderung
	TriggerStartF: F_TRIG;
	TriggerStopF	: F_TRIG;
	TriggerResetF : F_TRIG;
	TriggerStartR : R_TRIG;
	TriggerStopR : R_TRIG;
	TriggerResetR : R_TRIG;
	//Trigger NN-Änderungen
	Select_NN1_old	  : BOOL;
	Select_NN2_old	  : BOOL;

END_VAR

TriggerStartF(CLK := Start);
TriggerResetF(CLK := Reset);
TriggerStopF(CLK := Stop);
TriggerStartR(CLK := Start);
TriggerResetR(CLK := Reset);
TriggerStopR(CLK := Stop);

IF TriggerStartR.Q OR TriggerStartF.Q THEN
	CommunicationState := 1;
ELSIF TriggerStopR.Q OR TriggerStopF.Q THEN
	CommunicationState := 4;
ELSIF TriggerResetR.Q OR TriggerResetF.Q THEN
	CommunicationState := 5;
END_IF

CASE CommunicationState OF
	1:
		NewConfig := TRUE;
		IF Select_NN1 = Select_NN2 THEN
			Config_NN1 := Config_NN2 := FALSE;
		ELSE
			Config_NN1 := Select_NN1;
			Config_NN2 := Select_NN2;
		END_IF
		Select_NN1_old := Select_NN1;
		Select_NN2_old := Select_NN2;
		CommunicationState := 2;
	2:
		IF AcceptConfig THEN
			CommunicationState := 3;
			NewConfig := FALSE;
		END_IF
	3:
		Database[0] := X_Machine_CS;
		Database[1] := Y_Machine_CS;
		Database[2] := Z_Machine_CS;
		Database[3] := C_Machine_CS;
		Database[4] := B_Machine_CS;
		Database[5] := X_V_Machine_CS;
		Database[6] := Y_V_Machine_CS;
		Database[7] := Z_V_Machine_CS;
		Database[8] := C_V_Machine_CS;
		Database[9] := B_V_Machine_CS;
		Database[10] := n_Spindle;
		Database[11] := X_a_Machine_CS;
		Database[12] := Y_a_Machine_CS;
		Database[13] := Z_a_Machine_CS;
		Database[14] := C_a_Machine_CS;
		Database[15] := B_a_Machine_CS;
		Database[16] := n_a_Spindle;
		Database[17] := X_I;
		Database[18] := Y_I;
		Database[19] := Z_I;
		Database[20] := C_I;
		Database[21] := B_I;
		Database[22] := n_I;
		Database[23] := SIGNAL_FORCE[1];
		Database[24] := SIGNAL_FORCE[2];
		Database[25] := SIGNAL_FORCE[3];
		Database[26] := Depth;
		Database[27] := Width;

		yGraph1 := X_Machine_CS;
		yGraph2 := Y_Machine_CS;
		yGraph3 := Z_Machine_CS;
		Timer := Timer + (CycleTime / 100);
		
		DATA_PREPARATION ();
		
		IF Select_NN1_old <> Select_NN1_old OR Select_NN2_old <> Select_NN2 THEN
			CommunicationState := 1;
		END_IF
	4:
		Config_NN1 := FALSE;
		Config_NN2 := FALSE;
	5:
		FOR SetZeros := 0 TO 27 BY 1 DO
			Database[SetZeros] := 0 ;
		END_FOR;
		yGraph1 := yGraph2 := yGraph3 := 0;
		Config_NN1 := FALSE;
		Config_NN2 := FALSE;
		Timer := 0;
END_CASE;

END_PROGRAM

// ---- POUs/DATA_PREPARATION.TcPOU
PROGRAM DATA_PREPARATION
VAR	
	PrepPX :ARRAY[0..Buffersize] OF REAL;
	PrepPY :ARRAY[0..Buffersize] OF REAL;
	PrepPZ :ARRAY[0..Buffersize] OF REAL;
	PrepPC :ARRAY[0..Buffersize] OF REAL;
	PrepPB :ARRAY[0..Buffersize] OF REAL;
	PrepVX :ARRAY[0..Buffersize] OF REAL;
	PrepVY :ARRAY[0..Buffersize] OF REAL;
	PrepVZ :ARRAY[0..Buffersize] OF REAL;
	PrepVC :ARRAY[0..Buffersize] OF REAL;
	PrepVB :ARRAY[0..Buffersize] OF REAL;
	PrepVN :ARRAY[0..Buffersize] OF REAL;
	PrepAX :ARRAY[0..Buffersize] OF REAL;
	PrepAY :ARRAY[0..Buffersize] OF REAL;
	PrepAZ :ARRAY[0..Buffersize] OF REAL;
	PrepAC :ARRAY[0..Buffersize] OF REAL;
	PrepAB :ARRAY[0..Buffersize] OF REAL;
	PrepAN :ARRAY[0..Buffersize] OF REAL;
	PrepIX :ARRAY[0..Buffersize] OF REAL;
	PrepIY :ARRAY[0..Buffersize] OF REAL;
	PrepIZ :ARRAY[0..Buffersize] OF REAL;
	PrepIC :ARRAY[0..Buffersize] OF REAL;
	PrepIB :ARRAY[0..Buffersize] OF REAL;
	PrepIN :ARRAY[0..Buffersize] OF REAL;
	PrepF1 :ARRAY[0..Buffersize] OF REAL;
	PrepF2 :ARRAY[0..Buffersize] OF REAL;
	PrepF3 :ARRAY[0..Buffersize] OF REAL;
	
	Position_Counter :INT := 0;
	SumF1 : REAL := 0;
	SumF2 : REAL := 0;
	SumF3 : REAL := 0;
	
	{attribute 'OPC.UA.DA' := '1'}
	AverageF1 : REAL := 0;
	{attribute 'OPC.UA.DA' := '1'}
	AverageF2 : REAL := 0;
	{attribute 'OPC.UA.DA' := '1'}
	AverageF3 : REAL := 0;
END_VAR

VAR CONSTANT
	Buffersize : INT := 9;
END_VAR

FOR Position_Counter := Buffersize TO 1 BY -1 DO
	PrepF1[Position_Counter] := PrepF1[Position_Counter - 1];
	PrepF2[Position_Counter] := PrepF2[Position_Counter - 1];
	PrepF3[Position_Counter] := PrepF3[Position_Counter - 1];
END_FOR
FOR Position_Counter := Buffersize TO 0 BY -1 DO
	SumF1 := PrepF1[Position_Counter] + SumF1;
	SumF2 := PrepF2[Position_Counter] + SumF2;
	SumF3 := PrepF3[Position_Counter] + SumF3;
END_FOR
AverageF1 := SumF1 / (Buffersize + 1);
AverageF2 := SumF2 / (Buffersize + 1);
AverageF3 := SumF3 / (Buffersize + 1);
SumF1 := SumF2 := SumF3 := 0;

PrepF1[0] := Signal_Force[1];
PrepF2[0] := Signal_Force[2];
PrepF3[0] := Signal_Force[3];
Position_Counter := Buffersize;

END_PROGRAM

// ---- POUs/MEAS_STIFFNESS_COLLISION.TcPOU
PROGRAM MEAS_STIFFNESS_COLLISION
VAR
	
	//VARIABLES FOR STIFFNESS MEASUREMENT
	N_SAMPLES: WORD:=250;
	N_ACT: WORD;
	F1, F2, F3: REAL;
	P1, P2, P3: REAL;
	PROG_SYNCH: WORD;
	k: WORD:=0;
	
	
	
END_VAR


IF ACT_NC_PROGRAM=3 THEN		// MEASUREMENT OF TOOL STIFFNESS
	
	FORCE_ACT:=SIGNAL_FORCE_FLT[2];
	//FORCE_ACT:=A_SIGNAL_2;
	
	Y_POSITION_ACT:=ACT_NC_PARAM_5;			// in mm
	
		
	IF ACT_NC_PROGRAM_STEP=10 THEN
		F1:=0;
		F2:=0;
		F3:=0;
		P1:=0;
		P2:=0;
		P3:=0;
		N_ACT:=0;
		PROG_SYNCH:=1;
		FORCE_DEVIATION[1]:=0;
		COLLISION_DISTANCE:=0;
		TOOL_STIFFNESS[1]:=0;
		Z_POS_STIFF_MEAS[1]:=0;
		a_POS[1]:=0;
		TOOL_BLENDING_STIFFNESS[1]:=0;
	END_IF
	
	//GETTING Z POSITION FOR COLLISION
	IF ACT_NC_PROGRAM_STEP=20 THEN
		Z_POS_STIFF_MEAS[1]:=ACT_NC_PARAM_5;
	END_IF

	IF ACT_NC_PROGRAM_STEP=1 AND PROG_SYNCH=1 THEN
		F1:=F1+FORCE_ACT;
		P1:=P1+Y_POSITION_ACT;
		N_ACT:=N_ACT+1;
		IF N_ACT=N_SAMPLES THEN
			F1:=F1/N_SAMPLES;
			P1:=P1/N_SAMPLES;
			N_ACT:=0;
			PROG_SYNCH:=2;
		END_IF	
	END_IF

	IF ACT_NC_PROGRAM_STEP=2 AND PROG_SYNCH=2 THEN
		F2:=F2+FORCE_ACT;
		P2:=P2+Y_POSITION_ACT;
		N_ACT:=N_ACT+1;
		IF N_ACT=N_SAMPLES THEN
			F2:=F2/N_SAMPLES;
			P2:=P2/N_SAMPLES;
			N_ACT:=0;
			PROG_SYNCH:=3;
		END_IF	
	END_IF

	IF ACT_NC_PROGRAM_STEP=3 AND PROG_SYNCH=3 THEN
		F3:=F3+FORCE_ACT;
		P3:=P3+Y_POSITION_ACT;
		N_ACT:=N_ACT+1;
		IF N_ACT=N_SAMPLES THEN
			F3:=F3/N_SAMPLES;
			P3:=P3/N_SAMPLES;
			PROG_SYNCH:=0;
			FORCE_DEVIATION[1]:=(ABS(F2-F1)+ABS(F3-F2))/2;				// in N
			COLLISION_DISTANCE:=(ABS(P2-P1)+ABS(P3-P2))*1000/2; 	// in µm
			TOOL_STIFFNESS[1]:=FORCE_DEVIATION[1]/COLLISION_DISTANCE;		// in N/µm
			a_POS[1]:=TOOL_LENGTH-ABS(Z_POS_STIFF_MEAS[1])/2;				// in mm
			TOOL_BLENDING_STIFFNESS[1]:=FORCE_DEVIATION[1]*EXPT(a_POS[1],3)/3/COLLISION_DISTANCE*1000;	// in N.mm²
			a_REF:=TOOL_LENGTH-ABS(Z_POS_REF)/2;									   // in mm
			FOR k:=1 TO 5 BY 1 DO
				AX_SELC_PTS[k]:=TOOL_LENGTH-ABS(Z_POS_REF)+ABS(Z_POS_SELC_PTS[k]);
				IF AX_SELC_PTS[k]<=a_REF THEN
					TOOL_STIFFNESS_SELC_PTS[1,k]:=6*TOOL_BLENDING_STIFFNESS[1]/EXPT(AX_SELC_PTS[k],2)/(3*a_REF-AX_SELC_PTS[k])/1000; // in N/µm
				ELSE
					TOOL_STIFFNESS_SELC_PTS[1,k]:=6*TOOL_BLENDING_STIFFNESS[1]/EXPT(a_REF,2)/(3*AX_SELC_PTS[k]-a_REF)/1000; // in N/µm
				END_IF			
			END_FOR
		END_IF	
	END_IF
	
	

END_IF

END_PROGRAM

// ---- POUs/MEAS_STIFFNESS_PROCESS.TcPOU
PROGRAM MEAS_STIFFNESS_PROCESS
VAR
	
	//VARIABLES FOR STIFFNESS MEASUREMENT
	N_ACT_1: WORD;
	N_ACT_2: WORD;
	F1, F2: REAL;
	P1, P2: REAL;
	POS_LIM: ARRAY[1..4] OF REAL;
	k: WORD;
	
	
	
	
	
	
END_VAR

//MEASUREMENT OF TOOL STIFFNESS IN PROCESS
IF ACT_NC_PROGRAM=4 THEN		
	
	//CHOOSE FORCE SIGNAL
	FORCE_ACT:=SIGNAL_FORCE_FLT[2];
	//FORCE_ACT:=A_SIGNAL_2;
	X_POSITION_ACT:=ACT_NC_PARAM_5;		// in mm	
	
	//PROGRAM INITIALISATION		
	IF ACT_NC_PROGRAM_STEP=10 THEN
		F1:=0;
		F2:=0;
		P1:=0;
		P2:=0;
		N_ACT_1:=0;
		N_ACT_2:=0;
		FORCE_DEVIATION[2]:=0;
		SHAPE_DEVIATION:=0;
		TOOL_STIFFNESS[2]:=0;
		POS_LIM[1]:=0;
		POS_LIM[2]:=0;
		POS_LIM[3]:=0;
		POS_LIM[4]:=0;
		Z_POS_STIFF_MEAS[2]:=0;
		a_POS[2]:=0;
		TOOL_BLENDING_STIFFNESS[2]:=0;
	END_IF
	
	//GETTING POSITION RANGES/LIMITS FOR FORCE MEASURING
	IF ACT_NC_PROGRAM_STEP=20 THEN
		POS_LIM[1]:=ACT_NC_PARAM_5;
	END_IF
	
	IF ACT_NC_PROGRAM_STEP=21 THEN
		POS_LIM[2]:=ACT_NC_PARAM_5;
	END_IF
	
	IF ACT_NC_PROGRAM_STEP=22 THEN
		POS_LIM[3]:=ACT_NC_PARAM_5;
	END_IF
	
	IF ACT_NC_PROGRAM_STEP=23 THEN
		POS_LIM[4]:=ACT_NC_PARAM_5;
	END_IF
	
	//MEASURING Z POSITION, TAKE INTO ACCOUNT THE RADIUS OF THE TOUCH PROBE
	IF ACT_NC_PROGRAM_STEP=24 THEN
		Z_POS_STIFF_MEAS[2]:=ACT_NC_PARAM_5;
	END_IF
	 
	//PROGRAMATION BASED ON ONLINE AXIS POSITION INSTEAS OF DP RESETTING TO AVOID MILLING STOPS
	IF ACT_NC_PROGRAM_STEP=30 AND X_POSITION_ACT<POS_LIM[1] AND X_POSITION_ACT>POS_LIM[2] THEN
		F1:=F1+FORCE_ACT;
		N_ACT_1:=N_ACT_1+1;
	END_IF
	
	IF ACT_NC_PROGRAM_STEP=30 AND X_POSITION_ACT<POS_LIM[2] AND N_ACT_1>0  THEN
		F1:=F1/N_ACT_1;
		N_ACT_1:=0;
	END_IF	
	
	IF ACT_NC_PROGRAM_STEP=30 AND X_POSITION_ACT<POS_LIM[3] AND X_POSITION_ACT>POS_LIM[4] THEN
		F2:=F2+FORCE_ACT;
		N_ACT_2:=N_ACT_2+1;
	
	END_IF
	
	IF ACT_NC_PROGRAM_STEP=30 AND X_POSITION_ACT<POS_LIM[4] AND N_ACT_2>0  THEN
		F2:=F2/N_ACT_2;
		N_ACT_2:=0;
	END_IF
	
	//GETTING MESURED POSITION FROM TOUCH PROBE
	IF ACT_NC_PROGRAM_STEP=40 THEN
		P1:=ACT_NC_PARAM_5;
	END_IF	
	
	IF ACT_NC_PROGRAM_STEP=50 THEN
		P2:=ACT_NC_PARAM_5;
	END_IF

	//STIFFNESS CALCULATION
	IF 	ACT_NC_PROGRAM_STEP=60 THEN
		FORCE_DEVIATION[2]:=ABS(F2-F1);												// in N
		SHAPE_DEVIATION:=ABS(P2-P1)*1000;											// in µm
		TOOL_STIFFNESS[2]:=FORCE_DEVIATION[2]/SHAPE_DEVIATION;							// in N/µm
		a_POS[2]:=TOOL_LENGTH-ABS(Z_POS_STIFF_MEAS[2])/2;									// in mm
		TOOL_BLENDING_STIFFNESS[2]:=FORCE_DEVIATION[2]*EXPT(a_POS[2],3)/3/SHAPE_DEVIATION*1000;	// in N.mm² 
 		a_REF:=TOOL_LENGTH-ABS(Z_POS_REF)/2;									   // in mm
		FOR k:=1 TO 5 BY 1 DO
				AX_SELC_PTS[k]:=TOOL_LENGTH-ABS(Z_POS_REF)+ABS(Z_POS_SELC_PTS[k]);
				IF AX_SELC_PTS[k]<=a_REF THEN
					TOOL_STIFFNESS_SELC_PTS[2,k]:=6*TOOL_BLENDING_STIFFNESS[2]/EXPT(AX_SELC_PTS[k],2)/(3*a_REF-AX_SELC_PTS[k])/1000; // in N/µm
				ELSE
					TOOL_STIFFNESS_SELC_PTS[2,k]:=6*TOOL_BLENDING_STIFFNESS[2]/EXPT(a_REF,2)/(3*AX_SELC_PTS[k]-a_REF)/1000; // in N/µm
				END_IF			
		END_FOR
	END_IF

END_IF

END_PROGRAM

// ---- POUs/DEFLECTION_CONTROL_POSITION.TcPOU
PROGRAM DEFLECTION_CONTROL_POSITION
VAR
		USED_FORCE_SIGNAL: REAL:=0;
END_VAR

IF ACT_NC_PROGRAM=15 THEN
	
	//USED_FORCE_SIGNAL:=-A_SIGNAL_2;
	USED_FORCE_SIGNAL:=SIGNAL_FORCE_FLT[2];
	//USED_FORCE_SIGNAL:=SQRT(EXPT(A_SIGNAL_1,2)+EXPT(A_SIGNAL_2,2));
		
	IF USED_FORCE_SIGNAL<0 THEN
		FORCE_ACT:=0;
		ELSE FORCE_ACT:=USED_FORCE_SIGNAL;	
	END_IF
	
	(*IF ACT_NC_PROGRAM_STEP=11 THEN
		IF ACT_NC_PARAM_3=1 THEN
			TOOL_STIFFNESS_ACT:=TOOL_STIFFNESS_SELC_PTS[1,3];
			ELSE
			TOOL_STIFFNESS_ACT:=TOOL_STIFFNESS_SELC_PTS[2,3];
		END_IF
	END_IF
	
	IF ACT_NC_PROGRAM_STEP=12 THEN
		TOOL_STIFFNESS_ACT:=TOOL_STIFFNESS_SELC_PTS[2,3];
	END_IF
	*)
	//TOOL_STIFFNESS_ACT:=TOOL_STIFFNESS_SELC_PTS[1,3];
	//TOOL_STIFFNESS_ACT:=TOOL_STIFFNESS_SELC_PTS[2,3];
	TOOL_STIFFNESS_ACT:=6;  // Zur Sicherheit falls Steifigkeitsmessung nicht funktioniert
	DEFLECTION_ACT:=FORCE_ACT/TOOL_STIFFNESS_ACT;		//µm
		
	
	IF ACT_NC_PROGRAM_STEP=1 THEN
			DEFLECTION_CONTROL_ON:=1;			//DEFLECTION CONTROL ON		
		ELSE
			DEFLECTION_CONTROL_ON:=0;
	END_IF


	IF	DEFLECTION_CONTROL_ON=1 THEN
	
		//DEFLECTION_DIF:=DEFLECTION_REF-DEFLECTION_ACT;
		DEFLECTION_DIF:=-(0-DEFLECTION_ACT);
			
		POS_REG_P:=POS_K_P*DEFLECTION_DIF;
		POS_REG_I:=0;
		
		POS_REG:=POS_REG_P+POS_REG_I+POS_MID;
		POS_MACHINE:=POS_REG;
	
		IF POS_MACHINE > SATURATION_POS_MAX THEN
			POS_MACHINE:=SATURATION_POS_MAX;
		END_IF

		IF POS_MACHINE < SATURATION_POS_MIN THEN
			POS_MACHINE:=SATURATION_POS_MIN;
		END_IF
	
		ELSE POS_MACHINE:=POS_MID;
	
	END_IF
		
	SET_NC_PARAM_1:= REAL_TO_WORD(POS_MACHINE+1000);
	ELSE
		SET_NC_PARAM_1:= 1000;
END_IF

END_PROGRAM

// ---- POUs/ADAS_Kom.TcPOU
PROGRAM ADAS_Kom
VAR CONSTANT
	///defaultConfig : AdasConfiguration := (track := [1, 2, 3, 4, 5, 6, 7, 8, 9, 10, 11, 12, 13, 14, 15, 16, 17, 18, 19, 20, 21, 22, 23, 24, 25, 26, 27, 28, 29, 30],
	///										signal:= [4, 4, 4, 4, 4, 5, 5, 5, 5,  5,  5,  6,  6,  6,  6,  6,  6, 17, 17, 17, 17, 17, 17,  1,  1,  1,  1,  1,  1,  1],
	///										axis  := [1, 1, 2, 3, 4, 1, 1, 2, 3,  4,  5,  1,  1,  2,  3,  4,  5,  1,  1,  2,  3,  4,  5,  1,  1,  2,  3,  4,  5,  1]);
	///
	///
	///unten stehende Konfiguration nach neuen Schema
	///1->6
	///2->1
	///3->2
	///4->3
	///5->4
	///6->1
	///
	///											Messwert	Position		Geschwindigkeit				Beschleunigung				Strom						Offen
	///											Funktion x, x, x, x, o, 	x, x, x, x,  x,  ?,		 x,  x,  x,  x,  x,  ?,		 x,  x,  x,  x,  x,  ?,	
	///											Achse	 x, y, z, c, n, 	x, y, z, c,  b,  n, 	 x,  y,  z,  c,  b,  n,		 x,  y,  z,  c,  b,  n,
	defaultConfig: AdasConfiguration := (track := [1, 2, 3, 4, 5, 6, 7, 8, 9, 10, 11, 12, 13, 14, 15, 16, 17, 18, 19, 20, 21, 22, 23, 24, 25, 26, 27, 28, 29, 30], 
										signal := [4, 4, 4, 4, 4, 5, 5, 5, 5,  5,  5,  6,  6,  6,  6,  6,  6, 17, 17, 17, 17, 17, 17, 17,  4,  1,  1,  1,  1,  1], 
										  axis := [6, 1, 2, 3, 4, 6, 1, 2, 3,  4,  5,  6,  1,  2,  3,  4,  5,  6,  1,  2,  3,  4,  5,  6,  5,  6,  6,  1,  1,  1]);
	/// Lesen von allen 30 Datenstreams
	numberOfDefaultTracks: UINT := 30;
	/// Anzahl ms die nach Ausgabe einer Anforderung gewartet werden soll, bevor die Antwort ausgewertet wird.
	waitTime: INT := 50;
END_VAR
VAR_INPUT
	ADAS_IN AT %I*: ARRAY[0..63] OF WORD;
	/// UNION  aus DUTs
	adasStream_IN: AdasData_In;
	/// STRUCT aus DUTs
	requestedConfiguration_IN AT %I*: AdasConfiguration;
	numberOfRequestetTracks_IN AT %I*: UINT;
	ConfigRequest_IN AT %I*: BOOL;
END_VAR
VAR
	waitTimer: INT := 0;
	/// STRUCT aus DUTs
	actualConfig: AdasConfiguration;
	/// STRUCT aus DUTs
	requestedConfiguration: AdasConfiguration;
	configRequestTrigger: R_TRIG;
	tracksToConfig: UINT;
	configuredTracks: UINT := 0;
	index: UINT;
	///ENUM aus DUTs
	comState: eAdasKom_State := eAdasKom_State.WaitForNC;
	///ENUM aus DUTs
	configState: eAdasKonfig_State := eAdasKonfig_State.Init;
	selectCounter: SINT := 0;
	init: BOOL := 0;
	kommzeit: BOOL := 0;
	deint: BOOL := 0;
	track: BOOL := 0;
	signal: BOOL := 0;
END_VAR
VAR_OUTPUT
	/// UNION  aus DUTs
	adasStreamSetup_OUT AT %Q*: AdasSetup_Out;
	adasData AT %Q*: ARRAY[0..(gVarL.gVar_NumberOfAdasTracks - 1)] OF DINT;
	StartExe: INT;
END_VAR

adasStream_IN.asBin := ADAS_IN;

//Kommunikationszykluszeit von ADAS festlegen
IF kommzeit THEN
	//The machine axes numbers basically range from 1 to 31. Only axes that are enabled by 20070 $MC_AXCONF_MACHAX_USED within one of the active channels can supply data.
	adasStreamSetup_OUT.asSetup.blockType   := 15;	//entspricht 0xF aus Anleitung
	adasStreamSetup_OUT.asSetup.blockLength := 8;	//festgelegt in Anleitung
	adasStreamSetup_OUT.asSetup.selectTrack := 255; //Command mode
	adasStreamSetup_OUT.asSetup.selectAxis  := 100; //wenn man zykluszeit wechseln will
	adasStreamSetup_OUT.asSetup.selectSignal:= 8; //neue zykluszeit: 10x 0.5ms =5ms
	adasStreamSetup_OUT.asSetup.selectFlag  := adasStream_IN.asData.acceptFlag;
	kommzeit := 0;
	comState := eAdasKom_State.WaitForNC;
	configState := eAdasKonfig_State.Init;
END_IF


//Track bezeichnung senden von ADAS-Kommunikation
IF track THEN
	//The machine axes numbers basically range from 1 to 31. Only axes that are enabled by 20070 $MC_AXCONF_MACHAX_USED within one of the active channels can supply data.
	adasStreamSetup_OUT.asSetup.blockType   := 15;	//entspricht 0xF aus Anleitung
	adasStreamSetup_OUT.asSetup.blockLength := 8;	//festgelegt in Anleitung
	adasStreamSetup_OUT.asSetup.selectTrack := 255; //Comande mode
	adasStreamSetup_OUT.asSetup.selectAxis  := 122; //all tracks resetten
	adasStreamSetup_OUT.asSetup.selectSignal:= 0;   //Vorgabe
	adasStreamSetup_OUT.asSetup.selectFlag  := adasStream_IN.asData.acceptFlag;
	track := 0;
	comState := eAdasKom_State.WaitForNC;
	configState := eAdasKonfig_State.Init;
END_IF

//Signal bezeichnung senden von ADAS-Kommunikation
IF signal THEN
	//The machine axes numbers basically range from 1 to 31. Only axes that are enabled by 20070 $MC_AXCONF_MACHAX_USED within one of the active channels can supply data.
	adasStreamSetup_OUT.asSetup.blockType   := 15;	//entspricht 0xF aus Anleitung
	adasStreamSetup_OUT.asSetup.blockLength := 8;	//festgelegt in Anleitung
	adasStreamSetup_OUT.asSetup.selectTrack := 255; //Comande mode
	adasStreamSetup_OUT.asSetup.selectAxis  := 123; //all tracks resetten
	adasStreamSetup_OUT.asSetup.selectSignal:= 0;   //Vorgabe
	adasStreamSetup_OUT.asSetup.selectFlag  := adasStream_IN.asData.acceptFlag;
	signal := 0;
	comState := eAdasKom_State.WaitForNC;
//	configState := eAdasKonfig_State.Init;
END_IF


//Deinitialisierung von ADAS-Kommunikation
IF deint THEN
	//The machine axes numbers basically range from 1 to 31. Only axes that are enabled by 20070 $MC_AXCONF_MACHAX_USED within one of the active channels can supply data.
	adasStreamSetup_OUT.asSetup.blockType   := 15;	//entspricht 0xF aus Anleitung
	adasStreamSetup_OUT.asSetup.blockLength := 8;	//festgelegt in Anleitung
	adasStreamSetup_OUT.asSetup.selectTrack := 255; //Comande mode
	adasStreamSetup_OUT.asSetup.selectAxis  := 110; //all tracks resetten
	adasStreamSetup_OUT.asSetup.selectSignal:= 0;   //Vorgabe
	adasStreamSetup_OUT.asSetup.selectFlag  := adasStream_IN.asData.acceptFlag;
	deint := 0;
	comState := eAdasKom_State.WaitForNC;
	configState := eAdasKonfig_State.Init;
END_IF

//Initialisierung von ADAS-Kommunikation
IF init THEN
	//The machine axes numbers basically range from 1 to 31. Only axes that are enabled by 20070 $MC_AXCONF_MACHAX_USED within one of the active channels can supply data.
	adasStreamSetup_OUT.asSetup.blockType   := 15;	//entspricht 0xF aus Anleitung
	adasStreamSetup_OUT.asSetup.blockLength := 8;	//festgelegt in Anleitung
	adasStreamSetup_OUT.asSetup.selectTrack := 0;
	adasStreamSetup_OUT.asSetup.selectAxis  := 0;
	adasStreamSetup_OUT.asSetup.selectSignal:= 0;
	adasStreamSetup_OUT.asSetup.selectFlag  := adasStream_IN.asData.acceptFlag;
	init := 0;
	comState := eAdasKom_State.WaitForNC;
	configState := eAdasKonfig_State.Init;
END_IF




CASE comState OF
	eAdasKom_State.WaitForNC:
		IF adasStream_IN.asData.comCycle > 0 THEN
			comState := eAdasKom_State.SetDefaultkonfig;
			requestedConfiguration := defaultConfig;
			tracksToConfig := numberOfDefaultTracks;
			configState := eAdasKonfig_State.SendTrackConfig;
			configuredTracks := 0;		
		END_IF
		
	eAdasKom_State.SetDefaultkonfig:
		CASE configState OF
			eAdasKonfig_State.SendTrackConfig:
			    selectCounter := adasStream_IN.asData.acceptFlag;
				selectCounter := selectCounter + 1;
				IF (selectCounter > 127) THEN
					selectCounter := 0;
				END_IF
				adasStreamSetup_OUT.asSetup.selectAxis 	:= requestedConfiguration.axis[configuredTracks];
				adasStreamSetup_OUT.asSetup.selectSignal:= requestedConfiguration.signal[configuredTracks];
				adasStreamSetup_OUT.asSetup.selectTrack	:= requestedConfiguration.track[configuredTracks];
				adasStreamSetup_OUT.asSetup.selectFlag	:= selectCounter;
				configState := eAdasKonfig_State.WaitForSelectFlag;
				waitTimer := 0;
			eAdasKonfig_State.WaitForSelectFlag:
				waitTimer := waitTimer + 1;
				IF (waitTimer >= waitTime)THEN
					IF (adasStream_IN.asData.acceptFlag = selectCounter)THEN
						
						actualConfig.axis[requestedConfiguration.track[configuredTracks] - 1]  := requestedConfiguration.axis[configuredTracks];
						actualConfig.signal[requestedConfiguration.track[configuredTracks]- 1] := requestedConfiguration.signal[configuredTracks];
						actualConfig.track[requestedConfiguration.track[configuredTracks] - 1] := requestedConfiguration.track[configuredTracks];
						
						configuredTracks := configuredTracks + 1;
						IF configuredTracks = tracksToConfig THEN
							comState :=	eAdasKom_State.Running;
							configState := eAdasKonfig_State.ConfigCurrent;
						ELSE
							configState := eAdasKonfig_State.SendTrackConfig;
						END_IF
	
					ELSIF (adasStream_IN.asData.acceptFlag < 0) THEN
						comState :=	eAdasKom_State.Error;		
					END_IF
				END_IF
		END_CASE
				
	eAdasKom_State.Running:
		adasData := adasStream_IN.asData.Data;
		CASE configState OF 
			eAdasKonfig_State.ConfigCurrent:
				configRequestTrigger(CLK := ConfigRequest_IN);
				IF configRequestTrigger.Q THEN
					requestedConfiguration := requestedConfiguration_IN;
					tracksToConfig := numberOfRequestetTracks_IN;
					configuredTracks := 0;
					configState := eAdasKonfig_State.SendTrackConfig;
				END_IF
			eAdasKonfig_State.SendTrackConfig:
				selectCounter := adasStream_IN.asData.acceptFlag;
				selectCounter := selectCounter + 1;
				IF (selectCounter > 127) THEN
					selectCounter := 0;
				END_IF
				adasStreamSetup_OUT.asSetup.selectAxis 	:= requestedConfiguration.axis[configuredTracks];
				adasStreamSetup_OUT.asSetup.selectSignal:= requestedConfiguration.signal[configuredTracks];
				adasStreamSetup_OUT.asSetup.selectTrack	:= requestedConfiguration.track[configuredTracks];
				adasStreamSetup_OUT.asSetup.selectFlag	:= selectCounter;
				configState := eAdasKonfig_State.WaitForSelectFlag;
			eAdasKonfig_State.WaitForSelectFlag:
				IF (adasStream_IN.asData.acceptFlag = selectCounter)THEN
					
					actualConfig.axis[requestedConfiguration.track[configuredTracks]]   := requestedConfiguration.axis[configuredTracks];
					actualConfig.signal[requestedConfiguration.track[configuredTracks]] := requestedConfiguration.signal[configuredTracks];
					actualConfig.track[requestedConfiguration.track[configuredTracks]]  := requestedConfiguration.track[configuredTracks];
					
					configuredTracks := configuredTracks + 1;
					IF configuredTracks = tracksToConfig THEN
						configState := eAdasKonfig_State.ConfigCurrent;
					ELSE
						configState := eAdasKonfig_State.SendTrackConfig;
					END_IF
				ELSIF (adasStream_IN.asData.acceptFlag < 0) THEN
					comState :=	eAdasKom_State.Error;		
				END_IF
		END_CASE
	eAdasKom_State.Error:	
END_CASE

END_PROGRAM

// ---- POUs/MAGNITUDESPECTRUM.TcPOU
PROGRAM MAGNITUDESPECTRUM

VAR CONSTANT	
    cInitSource			: ST_MA_MultiArray_InitPars 
							:= ( eTypeCode := eMA_TypeCode_LREAL, nDims := 1, aDimSizes := [cBufferLength]);	
END_VAR

VAR
	nSample				: UDINT;
	//nChnIndex			: UDINT;
	//aEl3632 AT %I*		: ARRAY[1..cOversamples] OF INT;	// Input from hardware e.g. EL3632  A_OVERSAMPLING_INPUT_1
	//A_OVERSAMPLING_INPUT_1 AT%I*: ARRAY[0..9] OF INT; // Sensor 1 X
	aBuffer				: ARRAY[1..cOversamples] OF LREAL;  // InputBuffer
					
	fbSource			:  FB_CMA_Source :=(	stInitPars := cInitSource, 
												nOwnID := eID_Source, 
												aDestIDs := [eID_PowSpec, eID_MagSpec],
												nResultBuffers := 5);	// Initialize source buffers
		(* Result buffers *)										
	aMagSpectrumResult	: ARRAY[1..cFFTResult] OF LREAL;	                    
    fbSinkMag			: FB_CMA_Sink := (nOwnID := eID_SinkMag);  
	
	aPowSpectrumResult	: ARRAY[1..cFFTResult] OF LREAL;	                    
    fbSinkPow			: FB_CMA_Sink := (nOwnID := eID_SinkPow);      
	//fbSink				:  FB_CMA_Sink	:= (	nOwnID := eID_Sink);
	
	nCountResults		: ULINT;
	bCalculate1			: BOOL;
	bCalculate2			: BOOL;
	(* RMS value calculation *)
	nChannel			: UDINT;
	fSum				: LREAL;
	fRmsValue_Mag		: LREAL;	
	fRmsValue_Pow		: LREAL;
	fPSDValue_Mag		: LREAL;
	fPSDValue_Pow		: LREAL;
	(* max amplitude calculation *)
	fMaxAmpl			: LREAL;
	nIdxOfMaxAmpl		: UDINT;		 // index of max amplitude in spectrum result array 
	(* frequency calculation *)
	fSampleTaskCycleTime: LREAL := 1; 	// ms
	fSampleRate			: LREAL; 		// Hz  ( sample rate = oversampling factor / cycle time )
	fResolution			: LREAL; 		// Hz/Idx
	fFrequency			: LREAL; 		// Hz	
	ResultArray			: ARRAY[1..4] OF LREAL;
	
	fbErrHist			: FB_HRErrHist; // error monitoring

END_VAR

//FOR nChnIndex := 1 TO cMaxChannels DO
	

(* input from EL3632 *)
FOR nSample := 1 TO cOversamples DO
	aBuffer[nSample] := INT_TO_LREAL(A_OVERSAMPLING_INPUT_1[nSample-1]);
END_FOR
				

// Call source to collect data
fbSource.Input1D( pDataIn 			:= ADR(aBuffer),
				  nDataInSize 		:= SIZEOF(aBuffer), 
				  eElementType 		:= eMA_TypeCode_LREAL,
				  nWorkDim 			:= 0,
				  pStartIndex		:= 0,
				  nOptionPars		:= cCMA_Option_MarkInterruption ); 
IF fbSource.bError THEN
	fbErrHist.AddError(bErr:=TRUE, hrErrCode:=fbSource.hrErrorCode, sErrSource:='MAGNITUDESPECTRUM.fbSource'); // error monitoring
	// ToDo: if error
END_IF

// Push results to sink
fbSinkMag.Output1D(	pDataOut 		:= ADR(aMagSpectrumResult), 
					nDataOutSize 	:= SIZEOF(aMagSpectrumResult), 
					eElementType 	:= eMA_TypeCode_LREAL, 
					nWorkDim 		:= 0,
					nElements		:= 0,
					pStartIndex 	:= 0,
					nOptionPars		:= 0,
					bNewResult		=> bCalculate1 );
IF fbSinkMag.bError THEN
	fbErrHist.AddError(bErr:=TRUE, hrErrCode:=fbSinkMag.hrErrorCode, sErrSource:='MAGNITUDESPECTRUM.fbSinkMag'); // error monitoring
	// ToDo: if error
END_IF

(* Push results to sink *)
fbSinkPow.Output1D(	pDataOut 		:= ADR(aPowSpectrumResult), 
					nDataOutSize 	:= SIZEOF(aPowSpectrumResult), 
					eElementType 	:= eMA_TypeCode_LREAL, 
					nWorkDim 		:= 0,
					nElements		:= 0,
					pStartIndex 	:= 0,
					nOptionPars		:= 0,
					bNewResult		=> bCalculate2 );
IF fbSinkPow.bError THEN
	fbErrHist.AddError(bErr:=TRUE, hrErrCode:=fbSinkPow.hrErrorCode, sErrSource:='MAGNITUDESPECTRUM.fbSinkPow'); // error monitoring
	// ToDo: if error
END_IF

IF cScaling = E_CM_ScalingType.eCM_PeakAmplitude THEN
	IF bCalculate1 THEN
		IF NOT LrealIsNaN(aMagSpectrumResult[1]) THEN
			// Calculate RMS value of signal
			fSum := 0;	
			FOR nChannel := 1 TO cFFTResult DO
				fSum := fSum + (aMagSpectrumResult[nChannel] * aMagSpectrumResult[nChannel]);
			END_FOR
			fRmsValue_Mag := SQRT(fSum);
			
			// Calculate max amplitude in spectrum
			fMaxAmpl := 0;
			FOR nChannel:=1 TO cFFTResult DO
				IF aMagSpectrumResult[nChannel] > fMaxAmpl THEN
					fMaxAmpl := aMagSpectrumResult[nChannel];
					nIdxOfMaxAmpl := nChannel;
				END_IF
			END_FOR
			// Calculate frequency for max amplitude [ frequency = index * (sample rate / FFT length) ]
			fSampleRate := cOversamples * (1000.0 / fSampleTaskCycleTime);
			fResolution := fSampleRate / cFFTLength;
			fFrequency := (nIdxOfMaxAmpl-1) * fResolution; // -1 to consider DC = 0*fResolution
		END_IF
	END_IF
	
	IF bCalculate2 THEN
		IF NOT LrealIsNaN(aPowSpectrumResult[1]) THEN
			// Calculate RMS value of signal
			fSum := 0;	
			FOR nChannel := 1 TO cFFTResult DO
				fSum := fSum + aPowSpectrumResult[nChannel];
			END_FOR
			fRmsValue_Pow := SQRT(fSum);
			
			// Calculate max amplitude in spectrum
			fMaxAmpl := 0;
			FOR nChannel:=1 TO cFFTResult DO
				IF aPowSpectrumResult[nChannel] > fMaxAmpl THEN
					fMaxAmpl := aPowSpectrumResult[nChannel];
					nIdxOfMaxAmpl := nChannel;
				END_IF
			END_FOR
			// Calculate frequency for max amplitude [ frequency = index * (sample rate / FFT length) ]
			fSampleRate := cOversamples * (1000.0 / fSampleTaskCycleTime);
			fResolution := fSampleRate / cFFTLength;
			fFrequency := (nIdxOfMaxAmpl-1) * fResolution; // -1 to consider DC = 0*fResolution
		END_IF
	END_IF
	// ToDo: if new result is ready
	ResultArray[1] := fFrequency;
	ResultArray[2] := GVarL.X_Machine_CS;
	ResultArray[3] := GVarL.Y_Machine_CS;
	ResultArray[4] := GVarL.Z_Machine_CS;
	
ELSIF cScaling = E_CM_ScalingType.eCM_PowerSpectralDensity THEN
	IF bCalculate1 THEN
		IF NOT LrealIsNaN(aMagSpectrumResult[1]) THEN
			fMaxAmpl := 0;
			FOR nChannel:=1 TO cFFTResult DO
				IF aMagSpectrumResult[nChannel] > fMaxAmpl THEN
					fMaxAmpl := aMagSpectrumResult[nChannel];
					nIdxOfMaxAmpl := nChannel;
				END_IF
			END_FOR
			fSampleRate := cOversamples * (1000.0 / fSampleTaskCycleTime);
			fResolution := fSampleRate / cFFTLength;
			fFrequency := (nIdxOfMaxAmpl-1) * fResolution; // -1 to consider DC = 0*fResolution
			fPSDValue_Mag := (fMaxAmpl * fMaxAmpl)/ fSampleRate ;
		END_IF
	END_IF
	
	IF bCalculate2 THEN
		IF NOT LrealIsNaN(aPowSpectrumResult[1]) THEN
			fMaxAmpl := 0;
			FOR nChannel:=1 TO cFFTResult DO
				IF aPowSpectrumResult[nChannel] > fMaxAmpl THEN
					fMaxAmpl := aPowSpectrumResult[nChannel];
					nIdxOfMaxAmpl := nChannel;
				END_IF
			END_FOR
			fSampleRate := cOversamples * (1000.0 / fSampleTaskCycleTime);
			fResolution := fSampleRate / cFFTLength;
			fFrequency := (nIdxOfMaxAmpl-1) * fResolution; // -1 to consider DC = 0*fResolution
			fPSDValue_Pow := fMaxAmpl/ fSampleRate ;
		END_IF
	END_IF
END_IF
//END_FOR

END_PROGRAM

// ---- POUs/Error Monitoring/FB_HRErrHist.TcPOU
FUNCTION_BLOCK FB_HRErrHist
(* v1.10
build up an error history consisting of two arrays and one index.
The index shows the actual array position. The last error id and the count for this id are saved in the arrays.
If an error id is the same as the previous input error the counter is increased. Otherwise the index is increased.
*)
VAR_INPUT
	bEdgeDetect	: BOOL;	(* FALSE: every input(bErr) is processed; TRUE: only rising edge of input is processed *)
END_VAR
VAR_OUTPUT
	nErrSum		: UINT;
	nErrIdx		: UINT; // error list index of last occured error (max. cHistLen)
	aErrList	: ARRAY[1..cHistLen] OF ST_HRErrHist;
END_VAR

VAR
	bNewErr		: BOOL;
	fbErrTrig	: R_TRIG;
END_VAR
VAR CONSTANT
	cHistLen	: UINT := 100;
END_VAR

METHOD AddError
VAR_INPUT
	bErr		: BOOL;
	hrErrCode	: HRESULT;
	sErrSource	: STRING(63);
END_VAR
fbErrTrig(CLK:=bErr);
IF bEdgeDetect THEN
	bNewErr := fbErrTrig.Q;
ELSE
	bNewErr := bErr;
END_IF

IF bNewErr THEN
	nErrSum := nErrSum + 1;
	IF nErrIdx < cHistLen THEN
		IF nErrIdx = 0 THEN
			nErrIdx	:= nErrIdx + 1;
		ELSIF aErrList[nErrIdx].hrErrCode <> hrErrCode OR aErrList[nErrIdx].sErrSource <> sErrSource THEN
			nErrIdx	:= nErrIdx + 1;
		END_IF
		aErrList[nErrIdx].hrErrCode := hrErrCode;
		aErrList[nErrIdx].sErrSource := sErrSource;
		aErrList[nErrIdx].nErrCount := aErrList[nErrIdx].nErrCount + 1;
	END_IF
END_IF
END_METHOD

METHOD Reset
VAR_INPUT
END_VAR
nErrSum := 0;
nErrIdx := 0;
MEMSET(ADR(aErrList),0,SIZEOF(aErrList));
END_METHOD

END_FUNCTION_BLOCK

// ---- POUs/ANALOG_OUTPUT_EL4134.TcPOU
PROGRAM ANALOG_OUTPUT_EL4134
VAR
END_VAR

END_PROGRAM

// ---- POUs/Function Generator/FB_FunctionGenerator.TcPOU
// generates a signal build up by the specified function type. v1.6
FUNCTION_BLOCK FB_FunctionGenerator
VAR_INPUT
	bEnable		: BOOL 	:= TRUE;	// set TRUE to generate the specified signal; set FALSE to reset the signal buffer
	fFrequency	: LREAL := 1000;	// in [Hz]
	fAmplitude	: LREAL := 1;
	fOffset		: LREAL	:= 0;	
	nDutyCycle	: UINT 	:= 50;		// in [%] (for pulse function)
	eFunction	: E_FunctionType := E_FunctionType.Sine;	
END_VAR
VAR_IN_OUT
	aSignal		: ARRAY[1..cOversamples] OF LREAL;
END_VAR
VAR_OUTPUT
	bError		: BOOL;
END_VAR

VAR
	bInit						: BOOL := TRUE;
	fbGetTaskIdx				: GETCURTASKINDEX;
	
	fLastFrequency				: LREAL;		// in [Hz]
	fLastAmplitude				: LREAL;
	fLastOffset					: LREAL;
	nLastDutyCycle				: UINT;
	eLastFunction				: E_FunctionType;
	
	nSamples					: UDINT;
	fCycleTime					: LREAL;		// in [s]
	fDelta						: LREAL;		// amplitude delta per sample
	fPhase						: LREAL;		// in [°]
	nSign						: INT := 1;		// 1 or -1
	fLastSignalValue			: LREAL;		// amplitude
	fPeriod						: LREAL;		// in [s]
	fAngularIncrement			: LREAL;		// in [°]
	fAngularIncrementPerCycle	: LREAL;		// in [°]
	fAngularIncrementPerSample	: LREAL;		// in [°]
	(* for modulated signal (carrier signal without offset) *)
	fCarrierFrequency					: LREAL := 500;	// in [Hz] (sine)
	fCarrierAmplitude					: LREAL := 1;
	fCarrierPeriod						: LREAL;		// in [s]
	fCarrierAngularIncrement			: LREAL;		// in [°]
	fCarrierAngularIncrementPerCycle	: LREAL;		// in [°]
	fCarrierAngularIncrementPerSample	: LREAL;		// in [°]
				
END_VAR

IF bEnable THEN
	IF fLastFrequency <> fFrequency THEN
		bInit := TRUE; // For automatic initializing
		fLastFrequency := fFrequency;
	END_IF
	IF fLastAmplitude <> fAmplitude THEN
		bInit := TRUE; // For automatic initializing
		fLastAmplitude := fAmplitude;
	END_IF
	IF fLastOffset <> fOffset THEN
		bInit := TRUE; // For automatic initializing
		fLastOffset := fOffset;
	END_IF
	IF nLastDutyCycle <> nDutyCycle THEN
		bInit := TRUE; // For automatic initializing
		nLastDutyCycle := nDutyCycle;
	END_IF
	IF eLastFunction <> eFunction THEN
		bInit := TRUE; // For automatic initializing
		eLastFunction := eFunction;
	END_IF
	IF bInit THEN
		// Get task info	
		fbGetTaskIdx();
		fCycleTime := UDINT_TO_LREAL(TwinCAT_SystemInfoVarList._TaskInfo[fbGetTaskIdx.index].CycleTime) (*100ns*) / (10.0 * 1000.0 * 1000.0);	
		fLastSignalValue := 0;
		nSign := 1;
		fAngularIncrement := 0;
		// Flush out old data
		MEMSET(ADR(aSignal), 0, SIZEOF(aSignal));
		IF fFrequency > 0 AND fCycleTime > 0 THEN		
			// Calculate period, increments per plc cycle, increment per oversample
			IF cOversamples > 0 THEN			
				IF eFunction = E_FunctionType.Sine THEN
					fPeriod := 1/fFrequency;
					fAngularIncrementPerCycle := 360*(fCycleTime/fPeriod);
					fAngularIncrementPerSample := fAngularIncrementPerCycle/cOversamples;
					// no phase adjustment
					bInit := FALSE;	
				ELSIF eFunction = E_FunctionType.Square	THEN
					fPeriod := 1/fFrequency;
					fAngularIncrementPerCycle  := 360*(fCycleTime/fPeriod);
					fAngularIncrementPerSample := fAngularIncrementPerCycle/cOversamples;
					fPhase := 0.5*360;
					bInit := FALSE;
				ELSIF eFunction = E_FunctionType.Pulse THEN
					fPeriod := 1/fFrequency;
					fAngularIncrementPerCycle  := 360*(fCycleTime/fPeriod);
					fAngularIncrementPerSample := fAngularIncrementPerCycle/cOversamples;
					IF nDutyCycle > 100 THEN
						nDutyCycle := 100;
					END_IF
					fPhase := (UDINT_TO_LREAL(nDutyCycle)/100)*360;
					bInit := FALSE;					
				ELSIF eFunction = E_FunctionType.Triangular THEN
					fPeriod := 1/fFrequency;				
					fAngularIncrementPerCycle  := 360*(fCycleTime/fPeriod);
					fAngularIncrementPerSample := fAngularIncrementPerCycle/cOversamples;
					fPhase := 0.5*360; 
					fDelta := 4*(fAmplitude/(360/fAngularIncrementPerSample));				
					bInit := FALSE;
				ELSIF eFunction = E_FunctionType.Sawtooth THEN
					fPeriod := 1/fFrequency;			
					fAngularIncrementPerCycle  := 360*(fCycleTime/fPeriod);		
					fAngularIncrementPerSample := fAngularIncrementPerCycle/cOversamples;
					fDelta := fAmplitude/(360/fAngularIncrementPerSample);
					bInit := FALSE;
				ELSIF eFunction = E_FunctionType.AM THEN
					fPeriod := 1/fFrequency;
					fAngularIncrementPerCycle := 360*(fCycleTime/fPeriod);
					fAngularIncrementPerSample := fAngularIncrementPerCycle/cOversamples;
					// no phase adjustment
					fCarrierPeriod := 1/fCarrierFrequency;
					fCarrierAngularIncrementPerCycle := 360*(fCycleTime/fCarrierPeriod);
					fCarrierAngularIncrementPerSample := fCarrierAngularIncrementPerCycle/cOversamples;				
					// no phase adjustment	
					bInit := FALSE;
				ELSE
					bError := TRUE;	
				END_IF
			ELSE
				bError := TRUE;
			END_IF
		ELSE
			bError := TRUE;
		END_IF
	END_IF
	
	// Enable function generator
	IF NOT bError THEN		
		CASE eFunction OF		
			// sine: typical for vibrations originating from rotating machine
			E_FunctionType.Sine: Sine();
			
			// square: mixed sine signals good for analyzing spectrum				
			E_FunctionType.Square: Square();
			
			// pulse: mixed sine signals good for analyzing spectrum				
			E_FunctionType.Pulse: Pulse();
	
			// sawtooth: ramp-type vibrations, continuously increasing			
			E_FunctionType.Sawtooth: Sawtooth();
		
			// triangular: mixed sine signals good for analyzing spectrum
			E_FunctionType.Triangular: Triangular();
		
			// amplitude modulation: typical for vibrations originating from gear-tooth failure or bearing faults
			// Carrier signal with own frequency and amplitude		
			E_FunctionType.AM: AM();				
		END_CASE
	END_IF
ELSE
	// Flush out old data
	MEMSET(ADR(aSignal), 0, SIZEOF(aSignal));
	
	bInit := TRUE;
	bError := FALSE;
END_IF

METHOD PRIVATE AM
VAR_INPUT
END_VAR
{warning disable C0371}

FOR nSamples := 1 TO cOversamples DO
	// base signal * carrier signal
	aSignal[nSamples] := ( fAmplitude*SIN(2*PI*(fAngularIncrement+(nSamples-1)*fAngularIncrementPerSample)/360) + fOffset )
							* ( fCarrierAmplitude*SIN(2*PI*(fCarrierAngularIncrement+(nSamples-1)*fCarrierAngularIncrementPerSample)/360) );
END_FOR
// Increment angular positions
fAngularIncrement := fAngularIncrement + fAngularIncrementPerCycle;
fCarrierAngularIncrement := fCarrierAngularIncrement + fCarrierAngularIncrementPerCycle;

{warning restore C0371}
END_METHOD

METHOD PRIVATE Pulse
VAR_INPUT
END_VAR
{warning disable C0371}

FOR nSamples := 1 TO cOversamples DO
	// For pulse wave (unequal phases)
	IF (fAngularIncrement >= 360) THEN
		fAngularIncrement := fAngularIncrement - DINT_TO_LREAL(LREAL_TO_DINT(fAngularIncrement/360))*360;
		// or with Tc2_Math library: fAngularIncrement := LMOD(fAngularIncrement,360);
	END_IF
	IF (fAngularIncrement < fPhase) THEN
		nSign := 1;		
	ELSIF (fAngularIncrement >= fPhase) THEN
		nSign := 0;
	END_IF
	fAngularIncrement := fAngularIncrement + fAngularIncrementPerSample;
	
	aSignal[nSamples] := nSign*fAmplitude;
	
	aSignal[nSamples] := aSignal[nSamples] + fOffset;
END_FOR

{warning restore C0371}
END_METHOD

METHOD PRIVATE Sawtooth
VAR_INPUT
END_VAR
{warning disable C0371}

FOR nSamples := 1 TO cOversamples DO
	// For sawtooth wave (equal phase = period/2)
	IF (fAngularIncrement >= 360) THEN
		fAngularIncrement := fAngularIncrement - DINT_TO_LREAL(LREAL_TO_DINT(fAngularIncrement/360))*360;
		// or with Tc2_Math library: fAngularIncrement := LMOD(fAngularIncrement,360);
		fLastSignalValue := fLastSignalValue -fAmplitude;
	END_IF
	fAngularIncrement := fAngularIncrement + fAngularIncrementPerSample;

	aSignal[nSamples] := fLastSignalValue + fDelta;

	// Store last sample
	fLastSignalValue := aSignal[nSamples];
	
	aSignal[nSamples] := aSignal[nSamples] + fOffset;					
END_FOR	

{warning restore C0371}
END_METHOD

METHOD PRIVATE Sine
VAR_INPUT
END_VAR
{warning disable C0371}

FOR nSamples := 1 TO cOversamples DO
	aSignal[nSamples] := fAmplitude*SIN(2*PI*(fAngularIncrement+(nSamples-1)*fAngularIncrementPerSample)/360);

	aSignal[nSamples] := aSignal[nSamples] + fOffset;
END_FOR

// Increment angular position
fAngularIncrement := fAngularIncrement + fAngularIncrementPerCycle;

{warning restore C0371}
END_METHOD

METHOD PRIVATE Square
VAR_INPUT
END_VAR
{warning disable C0371}

FOR nSamples := 1 TO cOversamples DO
	// For square wave (equal phase = period/2)
	IF (fAngularIncrement >= 360) THEN
		fAngularIncrement := fAngularIncrement - DINT_TO_LREAL(LREAL_TO_DINT(fAngularIncrement/360))*360;
		// or with Tc2_Math library: fAngularIncrement := LMOD(fAngularIncrement,360);
	END_IF
	IF (fAngularIncrement < fPhase) THEN
		nSign := 1;
	ELSIF (fAngularIncrement >= fPhase) THEN
		nSign := -1;
	END_IF
	fAngularIncrement := fAngularIncrement + fAngularIncrementPerSample;
	
	aSignal[nSamples] := nSign*fAmplitude;
	
	aSignal[nSamples] := aSignal[nSamples] + fOffset;
END_FOR

{warning restore C0371}
END_METHOD

METHOD PRIVATE Triangular
VAR_INPUT
END_VAR
{warning disable C0371}

FOR nSamples := 1 TO cOversamples DO
	IF (fAngularIncrement >= 360) THEN
		fAngularIncrement := fAngularIncrement - DINT_TO_LREAL(LREAL_TO_DINT(fAngularIncrement/360))*360;
		// or with Tc2_Math library: fAngularIncrement := LMOD(fAngularIncrement,360);
	END_IF
	// Negative delta -> Positive delta
	IF fAngularIncrement < fPhase/2 THEN	
		nSign := 1;		
	ELSIF fAngularIncrement >= fPhase/2 AND fAngularIncrement < 3*fPhase/2 THEN
		nSign := -1;
	ELSIF fAngularIncrement >= 3*fPhase/2 THEN
		nSign := 1;	
	END_IF
	fAngularIncrement := fAngularIncrement + fAngularIncrementPerSample;
	
	aSignal[nSamples] := fLastSignalValue + nSign*fDelta;
	IF aSignal[nSamples] > fAmplitude THEN
		aSignal[nSamples] := aSignal[nSamples] - 2*(aSignal[nSamples]-fAmplitude);
	ELSIF aSignal[nSamples] < (-1)*fAmplitude THEN
		aSignal[nSamples] := aSignal[nSamples] - 2*(aSignal[nSamples]+fAmplitude);
	END_IF
	
	// Store last sample
	fLastSignalValue := aSignal[nSamples];		
	
	aSignal[nSamples] := aSignal[nSamples] + fOffset;
END_FOR

{warning restore C0371}
END_METHOD

END_FUNCTION_BLOCK

// ---- POUs/MAIN_CM.TcPOU
PROGRAM MAIN_CM

VAR CONSTANT
	cInitMagSpec 	: ST_CM_MagnitudeSpectrum_InitPars := (	nFFT_Length := cFFTLength, 
															nWindowLength := cWindowLength,
															bTransformToDecibel:= FALSE, 
															eWindowType := E_CM_WindowType.eCM_HannWindow,	
															eScalingType := E_CM_ScalingType.eCM_PeakAmplitude);	
															//fDecibelThreshold := cCM_MinArgLog10,
															//bTransformToDecibel := cDecibelScale,

	cInitPowSpec	: ST_CM_PowerSpectrum_InitPars :=  (	nFFT_Length := cFFTLength, 
															nWindowLength := cWindowLength,
															bTransformToDecibel:= FALSE,
															eWindowType := E_CM_WindowType.eCM_HannWindow,	
															eScalingType := eCM_PowerSpectralDensity);
															//fDecibelThreshold := cCM_MinArgLog10,
															//bTransformToDecibel := cDecibelScale,				
											
	// change eScalingType to E_CM_ScalingType.eCM_PeakAmplitude if max of spectrum has to be the amplitude value of a sine-wave
														
END_VAR

VAR	
														
	fbMagSpec			: FB_CMA_MagnitudeSpectrum :=(	stInitPars := cInitMagSpec, 
												nOwnID := eID_MagSpec, 
												aDestIDs := [eID_SinkMag],
												nResultBuffers   := 4);	

	fbPowSpec			: FB_CMA_PowerSpectrum :=(	stInitPars := cInitPowSpec, 
												nOwnID := eID_PowSpec, 
												aDestIDs := [eID_SinkPow],
												nResultBuffers   := 4);		
	fbErrHist			: FB_HRErrHist; // error monitoring
END_VAR

// Call Magnitude Spectrum 
fbMagSpec.Call();
IF fbMagSpec.bError THEN
	fbErrHist.AddError(bErr:=TRUE, hrErrCode:=fbMagSpec.hrErrorCode, sErrSource:='MAIN_CM.fbMagSpec'); // error monitoring
	// ToDo: if error
END_IF


// Call Power Spectrum 
fbPowSpec.Call();
IF fbPowSpec.bError THEN
	fbErrHist.AddError(bErr:=TRUE, hrErrCode:=fbPowSpec.hrErrorCode, sErrSource:='MAIN_CM.fbPowSpec'); // error monitoring
	// ToDo: if error
END_IF

END_PROGRAM

// ---- POUs/Test.TcPOU
PROGRAM Test
VAR
	
t : REAL:=0;
Y : REAL:=0;
Tsa : REAL:=0.004;
A : REAL:=0.1;
Control : WORD:=0;
F_sch: REAL:=1;
Vari: REAL:=0;
END_VAR

t:=t+Tsa;
Y:=A*SIN(2*3.14*F_sch*t); //mm

SET_NC_PARAM_1:=0;

IF Control=1 THEN
//SET_NC_PARAM_1:= REAL_TO_WORD(ABS(1000*Y));
SET_NC_PARAM_1:= REAL_TO_WORD(1000*(Y+A));
//Vari:=SET_NC_PARAM_1-*0.001;
(*SET_NC_PARAM_2:=1;
	IF Y<0 THEN 
		SET_NC_PARAM_2:=-1;
	END_IF
	*)
END_IF

END_PROGRAM

// ---- GlobalTextList.TcGTLO
TEXTLIST GlobalTextList
  830 = '%1u'
  186 = '%2x'
  617 = '%3f'
  832 = '%3u'
  543 = '00'
  292 = '01'
  293 = '02'
  294 = '03'
  295 = '04'
  296 = '05'
  298 = '06'
  299 = '07'
  846 = '08'
  847 = '09'
  297 = '1'
  848 = '10'
  381 = 'B0'
  382 = 'B1'
  383 = 'B2'
  384 = 'B3'
  385 = 'B4'
  386 = 'B5'
  387 = 'B6'
  388 = 'B7'
  389 = 'CAN Frame'
  618 = 'Collision distance [µm]'
  968 = 'Control off'
  967 = 'Control on'
  971 = 'Deflection control'
  608 = 'Deflection control off'
  972 = 'Deflection control on'
  834 = 'Downsampling NDS'
  619 = 'Force deviation [N]'
  614 = 'Force reset'
  187 = 'HUB'
  390 = 'ID'
  825 = 'NM / Frame'
  391 = 'Node'
  826 = 'NS / Meas'
  829 = 'Reset'
  544 = 'S1'
  393 = 'S10'
  545 = 'S2'
  546 = 'S3'
  547 = 'S4'
  548 = 'S5'
  549 = 'S6'
  550 = 'S7'
  379 = 'S8'
  380 = 'S9'
  185 = 'Send HUB-Frame'
  831 = 'Sensor Control'
  849 = 'Sensor Positions'
  613 = 'Sensor reset'
  611 = 'Sensor start'
  612 = 'Sensor stop'
  969 = 'Shape deviation [µm]'
  184 = 'Signal Noise'
  827 = 'Start'
  392 = 'State'
  616 = 'Stiffness measurement'
  828 = 'Stop'
  615 = 'System Control'
  970 = 'Test Setup'
  620 = 'Tool stiffness [N/µm]'
  833 = 'Trigger'
  609 = 'Trigger start'
  610 = 'Trigger stop'
END_TEXTLIST

// ---- VISUs/Datamodule.TcVIS
VISUALIZATION Datamodule  // 2x2
END_VISUALIZATION

// ---- VISUs/VISUALISATION_STIFFNESS_PROCESS.TcVIS
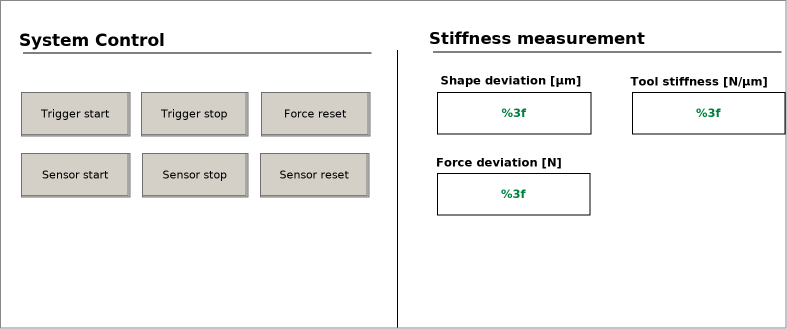
VISUALIZATION VISUALISATION_STIFFNESS_PROCESS  // 787x329
    Button (21,92 109x44), "Trigger start"
        OnMouseClick: execute { VARIABLES.CAN_TRIGGER_STATE:=1; }
    Button (141,92 107x44), "Trigger stop"
        OnMouseClick: execute { VARIABLES.CAN_TRIGGER_STATE:=0; }
    Button (21,153 109x44), "Sensor start"
        OnMouseClick: execute { CAN_CONTROL_STATE:=1; }
    Button (142,153 106x44), "Sensor stop"
        OnMouseClick: execute { CAN_CONTROL_STATE:=0; }
    Button (260,153 109x44), "Sensor reset"
        OnMouseClick: execute { CAN_CONTROL_STATE:=2; }
    Button (261,92 109x44), "Force reset"
        OnMouseClick: execute { VARIABLES.FORCE_RESET:=1; }
    Rectangle (17,25 150x30), "System Control"
    Line (371,53) (23,53)
    Rectangle (428,31 218x15), "Stiffness measurement"
    Rectangle (632,92 153x42), "%3f", text variable: VARIABLES.TOOL_STIFFNESS_SELC_PTS[2,3]
    Rectangle (437,92 154x42), "%3f", text variable: VARIABLES.SHAPE_DEVIATION
    Rectangle (437,173 153x42), "%3f", text variable: VARIABLES.FORCE_DEVIATION[2]
    Rectangle (437,73 148x15), "Shape deviation [µm]"
    Rectangle (437,155 124x15), "Force deviation [N]"
    Rectangle (632,74 135x15), "Tool stiffness [N/µm]"
    Line (397,50) (397,327)
    Line (781,52) (433,52)
END_VISUALIZATION
